LIN {X 0,Y 183.259,Z 699.514,A -85,B 0,C 180,E1 -22058.824,E2 -22058.824} C_VEL
LIN {X 0,Y 184.158,Z 697.784,A -85,B 0,C 180,E1 -22063.237,E2 -22063.237} C_VEL
LIN {X 0,Y 186.021,Z 694.918,A -85,B 0,C 180,E1 -22067.592,E2 -22067.592} C_VEL
LIN {X 0,Y 188.736,Z 690.854,A -85,B 0,C 180,E1 -22071.862,E2 -22071.862} C_VEL
LIN {X 0,Y 192.48,Z 685.477,A -85,B 0,C 180,E1 -22075.986,E2 -22075.986} C_VEL
LIN {X 0,Y 197.248,Z 678.651,A -85,B 0,C 180,E1 -22079.922,E2 -22079.922} C_VEL
LIN {X 0,Y 201.739,Z 671.619,A -85,B 0,C 180,E1 -22083.124,E2 -22083.124} C_VEL
LIN {X 0,Y 207.459,Z 662.596,A -85,B 0,C 180,E1 -22086.359,E2 -22086.359} C_VEL
LIN {X 0,Y 213.578,Z 652.129,A -85,B 0,C 180,E1 -22089.304,E2 -22089.304} C_VEL
LIN {X 0,Y 219.354,Z 641.413,A -85,B 0,C 180,E1 -22091.669,E2 -22091.669} C_VEL
LIN {X 0,Y 225.11,Z 629.438,A -85,B 0,C 180,E1 -22093.775,E2 -22093.775} C_VEL
LIN {X 0,Y 229.636,Z 618.5,A -85,B 0,C 180,E1 -22095.362,E2 -22095.362} C_VEL
LIN {X 0,Y 234.673,Z 604.884,A -85,B 0,C 180,E1 -22096.885,E2 -22096.885} C_VEL
LIN {X 0,Y 238.03,Z 593.851,A -85,B 0,C 180,E1 -22097.888,E2 -22097.888} C_VEL
LIN {X 0,Y 241.922,Z 578.93,A -85,B 0,C 180,E1 -22098.895,E2 -22098.895} C_VEL
LIN {X 0,Y 244.786,Z 564.165,A -85,B 0,C 180,E1 -22099.617,E2 -22099.617} C_VEL
LIN {X 0,Y 246.64,Z 549.204,A -85,B 0,C 180,E1 -22100.137,E2 -22100.137} C_VEL
LIN {X 0,Y 251.554,Z 483.18,A -85,B 0,C 180,E1 -22101.823,E2 -22101.823} C_VEL
LIN {X 0,Y 246.033,Z 470.679,A -85,B 0,C 180,E1 -22104.466,E2 -22104.466} C_VEL
LIN {X 0,Y 241.017,Z 460.608,A -85,B 0,C 180,E1 -22107.097,E2 -22107.097} C_VEL
LIN {X 0,Y 236.074,Z 451.47,A -85,B 0,C 180,E1 -22110.005,E2 -22110.005} C_VEL
LIN {X 0,Y 233.032,Z 446.227,A -85,B 0,C 180,E1 -22112.006,E2 -22112.006} C_VEL
LIN {X 0,Y 229.878,Z 441.234,A -85,B 0,C 180,E1 -22114.295,E2 -22114.295} C_VEL
LIN {X 0,Y 227.435,Z 437.174,A -85,B 0,C 180,E1 -22116.315,E2 -22116.315} C_VEL
LIN {X 0,Y 223.91,Z 432.279,A -85,B 0,C 180,E1 -22119.657,E2 -22119.657} C_VEL
LIN {X 0,Y 221.334,Z 429.386,A -85,B 0,C 180,E1 -22122.645,E2 -22122.645} C_VEL
LIN {X 0,Y 220.368,Z 427.276,A -85,B 0,C 180,E1 -22124.153,E2 -22124.153} C_VEL
LIN {X 0,Y 217.435,Z 424.585,A -85,B 0,C 180,E1 -22130.019,E2 -22130.019} C_VEL
LIN {X 0,Y 216.873,Z 422.233,A -85,B 0,C 180,E1 -22133.722,E2 -22133.722} C_VEL
LIN {X 0,Y 217.021,Z 422.113,A -85,B 0,C 180,E1 -22137.712,E2 -22137.712} C_VEL
LIN {X 0,Y 218.644,Z 426.038,A -85,B 0,C 180,E1 -22143.478,E2 -22143.478} C_VEL
LIN {X 0,Y 220.595,Z 427.431,A -85,B 0,C 180,E1 -22146.633,E2 -22146.633} C_VEL
LIN {X 0,Y 222.451,Z 430.766,A -85,B 0,C 180,E1 -22149.219,E2 -22149.219} C_VEL
LIN {X 0,Y 224.481,Z 432.884,A -85,B 0,C 180,E1 -22151.385,E2 -22151.385} C_VEL
LIN {X 0,Y 227.136,Z 436.564,A -85,B 0,C 180,E1 -22153.876,E2 -22153.876} C_VEL
LIN {X 0,Y 228.488,Z 438.495,A -85,B 0,C 180,E1 -22155.014,E2 -22155.014} C_VEL
LIN {X 0,Y 231.327,Z 442.468,A -85,B 0,C 180,E1 -22157.174,E2 -22157.174} C_VEL
LIN {X 0,Y 234.852,Z 447.543,A -85,B 0,C 180,E1 -22159.553,E2 -22159.553} C_VEL
LIN {X 0,Y 239.256,Z 453.973,A -85,B 0,C 180,E1 -22162.166,E2 -22162.166} C_VEL
LIN {X 0,Y 245.737,Z 464.47,A -85,B 0,C 180,E1 -22165.541,E2 -22165.541} C_VEL
LIN {X 0,Y 250.868,Z 473.742,A -85,B 0,C 180,E1 -22167.93,E2 -22167.93} C_VEL
LIN {X 0,Y 251.979,Z 476.143,A -85,B 0,C 180,E1 -22168.434,E2 -22168.434} C_VEL
LIN {X 0,Y 247.582,Z 533.829,A -85,B 0,C 180,E1 -22169.849,E2 -22169.849} C_VEL
LIN {X 0,Y 246.025,Z 550.183,A -85,B 0,C 180,E1 -22170.374,E2 -22170.374} C_VEL
LIN {X 0,Y 243.766,Z 564.236,A -85,B 0,C 180,E1 -22171.029,E2 -22171.029} C_VEL
LIN {X 0,Y 240.872,Z 577.724,A -85,B 0,C 180,E1 -22171.905,E2 -22171.905} C_VEL
LIN {X 0,Y 236.947,Z 591.791,A -85,B 0,C 180,E1 -22173.079,E2 -22173.079} C_VEL
LIN {X 0,Y 233.016,Z 603.642,A -85,B 0,C 180,E1 -22174.345,E2 -22174.345} C_VEL
LIN {X 0,Y 227.704,Z 617.399,A -85,B 0,C 180,E1 -22176.242,E2 -22176.242} C_VEL
LIN {X 0,Y 221.933,Z 629.908,A -85,B 0,C 180,E1 -22178.394,E2 -22178.394} C_VEL
LIN {X 0,Y 215.979,Z 641.386,A -85,B 0,C 180,E1 -22180.913,E2 -22180.913} C_VEL
LIN {X 0,Y 210.607,Z 650.717,A -85,B 0,C 180,E1 -22183.464,E2 -22183.464} C_VEL
LIN {X 0,Y 204.838,Z 659.969,A -85,B 0,C 180,E1 -22186.67,E2 -22186.67} C_VEL
LIN {X 0,Y 199.72,Z 667.593,A -85,B 0,C 180,E1 -22190.044,E2 -22190.044} C_VEL
LIN {X 0,Y 195.23,Z 673.844,A -85,B 0,C 180,E1 -22193.56,E2 -22193.56} C_VEL
LIN {X 0,Y 190.825,Z 679.701,A -85,B 0,C 180,E1 -22197.898,E2 -22197.898} C_VEL
LIN {X 0,Y 188.424,Z 682.875,A -85,B 0,C 180,E1 -22200.995,E2 -22200.995} C_VEL
LIN {X 0,Y 185.865,Z 686.124,A -85,B 0,C 180,E1 -22205.422,E2 -22205.422} C_VEL
LIN {X 0,Y 184.12,Z 688.111,A -85,B 0,C 180,E1 -22209.908,E2 -22209.908} C_VEL
LIN {X 0,Y 183.277,Z 688.904,A -85,B 0,C 180,E1 -22214.43,E2 -22214.43} C_VEL
LIN {X 0,Y 182.843,Z 688.545,A -85,B 0,C 180,E1 -22218.92,E2 -22218.92} C_VEL
LIN {X 0,Y 183.06,Z 687.039,A -85,B 0,C 180,E1 -22223.386,E2 -22223.386} C_VEL
LIN {X 0,Y 183.36,Z 685.852,A -85,B 0,C 180,E1 -22225.604,E2 -22225.604} C_VEL
LIN {X 0,Y 183.892,Z 682.596,A -85,B 0,C 180,E1 -22230,E2 -22230} C_VEL
LIN {X 0,Y 185.221,Z 678.05,A -85,B 0,C 180,E1 -22234.352,E2 -22234.352} C_VEL
LIN {X 0,Y 187.182,Z 672.165,A -85,B 0,C 180,E1 -22238.638,E2 -22238.638} C_VEL
LIN {X 0,Y 190.032,Z 664.763,A -85,B 0,C 180,E1 -22242.821,E2 -22242.821} C_VEL
LIN {X 0,Y 193.156,Z 656.84,A -85,B 0,C 180,E1 -22246.379,E2 -22246.379} C_VEL
LIN {X 0,Y 196.913,Z 647.341,A -85,B 0,C 180,E1 -22249.82,E2 -22249.82} C_VEL
LIN {X 0,Y 200.691,Z 637.648,A -85,B 0,C 180,E1 -22252.657,E2 -22252.657} C_VEL
LIN {X 0,Y 204.827,Z 626.148,A -85,B 0,C 180,E1 -22255.398,E2 -22255.398} C_VEL
LIN {X 0,Y 208.966,Z 613.481,A -85,B 0,C 180,E1 -22257.817,E2 -22257.817} C_VEL
LIN {X 0,Y 212.598,Z 600.987,A -85,B 0,C 180,E1 -22259.727,E2 -22259.727} C_VEL
LIN {X 0,Y 215.977,Z 587.405,A -85,B 0,C 180,E1 -22261.376,E2 -22261.376} C_VEL
LIN {X 0,Y 218.792,Z 573.543,A -85,B 0,C 180,E1 -22262.687,E2 -22262.687} C_VEL
LIN {X 0,Y 221.131,Z 558.77,A -85,B 0,C 180,E1 -22263.724,E2 -22263.724} C_VEL
LIN {X 0,Y 222.823,Z 543.551,A -85,B 0,C 180,E1 -22264.455,E2 -22264.455} C_VEL
LIN {X 0,Y 228.065,Z 457.657,A -85,B 0,C 180,E1 -22266.934,E2 -22266.934} C_VEL
LIN {X 0,Y 223.194,Z 447.442,A -85,B 0,C 180,E1 -22268.557,E2 -22268.557} C_VEL
LIN {X 0,Y 216.298,Z 434.861,A -85,B 0,C 180,E1 -22270.971,E2 -22270.971} C_VEL
LIN {X 0,Y 209.237,Z 423.431,A -85,B 0,C 180,E1 -22273.66,E2 -22273.66} C_VEL
LIN {X 0,Y 202.644,Z 414.059,A -85,B 0,C 180,E1 -22276.417,E2 -22276.417} C_VEL
LIN {X 0,Y 199.885,Z 410.222,A -85,B 0,C 180,E1 -22277.672,E2 -22277.672} C_VEL
LIN {X 0,Y 196.906,Z 406.254,A -85,B 0,C 180,E1 -22279.099,E2 -22279.099} C_VEL
LIN {X 0,Y 194.318,Z 402.919,A -85,B 0,C 180,E1 -22280.412,E2 -22280.412} C_VEL
LIN {X 0,Y 193.325,Z 401.554,A -85,B 0,C 180,E1 -22280.942,E2 -22280.942} C_VEL
LIN {X 0,Y 190.775,Z 398.797,A -85,B 0,C 180,E1 -22282.315,E2 -22282.315} C_VEL
LIN {X 0,Y 189.719,Z 396.646,A -85,B 0,C 180,E1 -22282.982,E2 -22282.982} C_VEL
LIN {X 0,Y 187.094,Z 394.663,A -85,B 0,C 180,E1 -22284.473,E2 -22284.473} C_VEL
LIN {X 0,Y 185.803,Z 392.386,A -85,B 0,C 180,E1 -22285.349,E2 -22285.349} C_VEL
LIN {X 0,Y 185.5,Z 390.99,A -85,B 0,C 180,E1 -22285.684,E2 -22285.684} C_VEL
LIN {X 0,Y 185.524,Z 390.96,A -85,B 0,C 180,E1 -22290.609,E2 -22290.609} C_VEL
LIN {X 0,Y 185.547,Z 390.93,A -85,B 0,C 180,E1 -22295.376,E2 -22295.376} C_VEL
LIN {X 0,Y 185.636,Z 390.969,A -85,B 0,C 180,E1 -22301.17,E2 -22301.17} C_VEL
LIN {X 0,Y 185.673,Z 390.975,A -85,B 0,C 180,E1 -22304.634,E2 -22304.634} C_VEL
LIN {X 0,Y 185.89,Z 390.93,A -85,B 0,C 180,E1 -22309.418,E2 -22309.418} C_VEL
LIN {X 0,Y 185.934,Z 390.931,A -85,B 0,C 180,E1 -22313.488,E2 -22313.488} C_VEL
LIN {X 0,Y 186.179,Z 390.916,A -85,B 0,C 180,E1 -22317.836,E2 -22317.836} C_VEL
LIN {X 0,Y 186.383,Z 390.877,A -85,B 0,C 180,E1 -22319.999,E2 -22319.999} C_VEL
LIN {X 0,Y 185.896,Z 390.952,A -85,B 0,C 180,E1 -22324.335,E2 -22324.335} C_VEL
LIN {X 0,Y 185.975,Z 390.929,A -85,B 0,C 180,E1 -22328.693,E2 -22328.693} C_VEL
LIN {X 0,Y 185.711,Z 390.958,A -85,B 0,C 180,E1 -22333.123,E2 -22333.123} C_VEL
LIN {X 0,Y 185.635,Z 390.971,A -85,B 0,C 180,E1 -22338.829,E2 -22338.829} C_VEL
LIN {X 0,Y 185.609,Z 390.984,A -85,B 0,C 180,E1 -22344.018,E2 -22344.018} C_VEL
LIN {X 0,Y 186.38,Z 393.478,A -85,B 0,C 180,E1 -22344.647,E2 -22344.647} C_VEL
LIN {X 0,Y 188.13,Z 395.653,A -85,B 0,C 180,E1 -22345.738,E2 -22345.738} C_VEL
LIN {X 0,Y 189.916,Z 396.943,A -85,B 0,C 180,E1 -22346.733,E2 -22346.733} C_VEL
LIN {X 0,Y 192.005,Z 400.303,A -85,B 0,C 180,E1 -22347.967,E2 -22347.967} C_VEL
LIN {X 0,Y 193.974,Z 402.192,A -85,B 0,C 180,E1 -22348.985,E2 -22348.985} C_VEL
LIN {X 0,Y 196.455,Z 405.732,A -85,B 0,C 180,E1 -22350.277,E2 -22350.277} C_VEL
LIN {X 0,Y 197.925,Z 407.506,A -85,B 0,C 180,E1 -22350.988,E2 -22350.988} C_VEL
LIN {X 0,Y 201.75,Z 412.692,A -85,B 0,C 180,E1 -22352.771,E2 -22352.771} C_VEL
LIN {X 0,Y 206.077,Z 418.936,A -85,B 0,C 180,E1 -22354.653,E2 -22354.653} C_VEL
LIN {X 0,Y 212.934,Z 431.449,A -85,B 0,C 180,E1 -22357.483,E2 -22357.483} C_VEL
LIN {X 0,Y 219.603,Z 445.413,A -85,B 0,C 180,E1 -22360.02,E2 -22360.02} C_VEL
LIN {X 0,Y 224.756,Z 457.578,A -85,B 0,C 180,E1 -22361.869,E2 -22361.869} C_VEL
LIN {X 0,Y 225.403,Z 459.29,A -85,B 0,C 180,E1 -22362.099,E2 -22362.099} C_VEL
LIN {X 0,Y 225.844,Z 462.305,A -85,B 0,C 180,E1 -22362.335,E2 -22362.335} C_VEL
LIN {X 0,Y 225.217,Z 466.845,A -85,B 0,C 180,E1 -22362.381,E2 -22362.381} C_VEL
LIN {X 0,Y 222.038,Z 477.484,A -85,B 0,C 180,E1 -22362.076,E2 -22362.076} C_VEL
LIN {X 0,Y 221.658,Z 480.258,A -85,B 0,C 180,E1 -22362.105,E2 -22362.105} C_VEL
LIN {X 0,Y 217.032,Z 553.649,A -85,B 0,C 180,E1 -22364.264,E2 -22364.264} C_VEL
LIN {X 0,Y 215.049,Z 569.791,A -85,B 0,C 180,E1 -22365.031,E2 -22365.031} C_VEL
LIN {X 0,Y 212.237,Z 585.232,A -85,B 0,C 180,E1 -22366.106,E2 -22366.106} C_VEL
LIN {X 0,Y 209.045,Z 599.111,A -85,B 0,C 180,E1 -22367.422,E2 -22367.422} C_VEL
LIN {X 0,Y 205.475,Z 612.527,A -85,B 0,C 180,E1 -22369.105,E2 -22369.105} C_VEL
LIN {X 0,Y 201.856,Z 623.921,A -85,B 0,C 180,E1 -22370.872,E2 -22370.872} C_VEL
LIN {X 0,Y 197.797,Z 635.793,A -85,B 0,C 180,E1 -22373.159,E2 -22373.159} C_VEL
LIN {X 0,Y 193.573,Z 646.785,A -85,B 0,C 180,E1 -22375.753,E2 -22375.753} C_VEL
LIN {X 0,Y 189.625,Z 656.949,A -85,B 0,C 180,E1 -22378.743,E2 -22378.743} C_VEL
LIN {X 0,Y 185.641,Z 666.861,A -85,B 0,C 180,E1 -22382.37,E2 -22382.37} C_VEL
LIN {X 0,Y 182.276,Z 675.104,A -85,B 0,C 180,E1 -22386.118,E2 -22386.118} C_VEL
LIN {X 0,Y 179.877,Z 681.389,A -85,B 0,C 180,E1 -22389.668,E2 -22389.668} C_VEL
LIN {X 0,Y 177.864,Z 687.458,A -85,B 0,C 180,E1 -22393.943,E2 -22393.943} C_VEL
LIN {X 0,Y 176.556,Z 692.457,A -85,B 0,C 180,E1 -22398.52,E2 -22398.52} C_VEL
LIN {X 0,Y 176.035,Z 696.126,A -85,B 0,C 180,E1 -22403.121,E2 -22403.121} C_VEL
LIN {X 0,Y 176.019,Z 698.545,A -85,B 0,C 180,E1 -22407.712,E2 -22407.712} C_VEL
LIN {X 0,Y 176.131,Z 699.306,A -85,B 0,C 180,E1 -22410,E2 -22410} C_VEL
LIN {X 0,Y 175.936,Z 699.898,A -85,B 0,C 180,E1 -22414.582,E2 -22414.582} C_VEL
LIN {X 0,Y 176.214,Z 699.33,A -85,B 0,C 180,E1 -22419.18,E2 -22419.18} C_VEL
LIN {X 0,Y 177.194,Z 697.647,A -85,B 0,C 180,E1 -22423.767,E2 -22423.767} C_VEL
LIN {X 0,Y 179.196,Z 694.83,A -85,B 0,C 180,E1 -22428.286,E2 -22428.286} C_VEL
LIN {X 0,Y 182.121,Z 690.816,A -85,B 0,C 180,E1 -22432.699,E2 -22432.699} C_VEL
LIN {X 0,Y 186.067,Z 685.473,A -85,B 0,C 180,E1 -22436.953,E2 -22436.953} C_VEL
LIN {X 0,Y 191.084,Z 678.704,A -85,B 0,C 180,E1 -22440.992,E2 -22440.992} C_VEL
LIN {X 0,Y 196.799,Z 670.339,A -85,B 0,C 180,E1 -22444.847,E2 -22444.847} C_VEL
LIN {X 0,Y 202.654,Z 661.439,A -85,B 0,C 180,E1 -22447.993,E2 -22447.993} C_VEL
LIN {X 0,Y 208.138,Z 652.404,A -85,B 0,C 180,E1 -22450.541,E2 -22450.541} C_VEL
LIN {X 0,Y 214.113,Z 641.786,A -85,B 0,C 180,E1 -22452.929,E2 -22452.929} C_VEL
LIN {X 0,Y 220.036,Z 629.994,A -85,B 0,C 180,E1 -22455.036,E2 -22455.036} C_VEL
LIN {X 0,Y 224.731,Z 619.14,A -85,B 0,C 180,E1 -22456.644,E2 -22456.644} C_VEL
LIN {X 0,Y 229.904,Z 605.716,A -85,B 0,C 180,E1 -22458.17,E2 -22458.17} C_VEL
LIN {X 0,Y 233.366,Z 594.831,A -85,B 0,C 180,E1 -22459.171,E2 -22459.171} C_VEL
LIN {X 0,Y 237.343,Z 580.285,A -85,B 0,C 180,E1 -22460.178,E2 -22460.178} C_VEL
LIN {X 0,Y 240.466,Z 565.248,A -85,B 0,C 180,E1 -22460.926,E2 -22460.926} C_VEL
LIN {X 0,Y 242.522,Z 549.652,A -85,B 0,C 180,E1 -22461.484,E2 -22461.484} C_VEL
LIN {X 0,Y 247.411,Z 486.673,A -85,B 0,C 180,E1 -22463.089,E2 -22463.089} C_VEL
LIN {X 0,Y 247.105,Z 485.359,A -85,B 0,C 180,E1 -22463.269,E2 -22463.269} C_VEL
LIN {X 0,Y 242.127,Z 473.926,A -85,B 0,C 180,E1 -22465.83,E2 -22465.83} C_VEL
LIN {X 0,Y 237.321,Z 464.186,A -85,B 0,C 180,E1 -22468.542,E2 -22468.542} C_VEL
LIN {X 0,Y 233.344,Z 456.624,A -85,B 0,C 180,E1 -22471.06,E2 -22471.06} C_VEL
LIN {X 0,Y 230.817,Z 452.144,A -85,B 0,C 180,E1 -22472.825,E2 -22472.825} C_VEL
LIN {X 0,Y 227.468,Z 446.57,A -85,B 0,C 180,E1 -22475.425,E2 -22475.425} C_VEL
LIN {X 0,Y 225.593,Z 443.377,A -85,B 0,C 180,E1 -22477.082,E2 -22477.082} C_VEL
LIN {X 0,Y 222.514,Z 438.986,A -85,B 0,C 180,E1 -22480.152,E2 -22480.152} C_VEL
LIN {X 0,Y 220.034,Z 436.054,A -85,B 0,C 180,E1 -22483.18,E2 -22483.18} C_VEL
LIN {X 0,Y 219.112,Z 434.167,A -85,B 0,C 180,E1 -22484.674,E2 -22484.674} C_VEL
LIN {X 0,Y 216.43,Z 431.406,A -85,B 0,C 180,E1 -22490.486,E2 -22490.486} C_VEL
LIN {X 0,Y 215.965,Z 429.13,A -85,B 0,C 180,E1 -22494.398,E2 -22494.398} C_VEL
LIN {X 0,Y 216.147,Z 429.172,A -85,B 0,C 180,E1 -22497.703,E2 -22497.703} C_VEL
LIN {X 0,Y 217.54,Z 432.906,A -85,B 0,C 180,E1 -22503.028,E2 -22503.028} C_VEL
LIN {X 0,Y 219.466,Z 434.461,A -85,B 0,C 180,E1 -22506.321,E2 -22506.321} C_VEL
LIN {X 0,Y 221.456,Z 437.897,A -85,B 0,C 180,E1 -22509.131,E2 -22509.131} C_VEL
LIN {X 0,Y 223.066,Z 439.594,A -85,B 0,C 180,E1 -22510.898,E2 -22510.898} C_VEL
LIN {X 0,Y 225.595,Z 443.212,A -85,B 0,C 180,E1 -22513.37,E2 -22513.37} C_VEL
LIN {X 0,Y 229.559,Z 449.003,A -85,B 0,C 180,E1 -22516.623,E2 -22516.623} C_VEL
LIN {X 0,Y 233.234,Z 454.435,A -85,B 0,C 180,E1 -22519.187,E2 -22519.187} C_VEL
LIN {X 0,Y 238.216,Z 462.153,A -85,B 0,C 180,E1 -22522.211,E2 -22522.211} C_VEL
LIN {X 0,Y 243.893,Z 471.728,A -85,B 0,C 180,E1 -22525.225,E2 -22525.225} C_VEL
LIN {X 0,Y 247.906,Z 479.45,A -85,B 0,C 180,E1 -22527.175,E2 -22527.175} C_VEL
LIN {X 0,Y 242.697,Z 544.089,A -85,B 0,C 180,E1 -22528.784,E2 -22528.784} C_VEL
LIN {X 0,Y 240.794,Z 558.358,A -85,B 0,C 180,E1 -22529.38,E2 -22529.38} C_VEL
LIN {X 0,Y 238.341,Z 570.495,A -85,B 0,C 180,E1 -22530.021,E2 -22530.021} C_VEL
LIN {X 0,Y 234.86,Z 584.57,A -85,B 0,C 180,E1 -22531.065,E2 -22531.065} C_VEL
LIN {X 0,Y 230.657,Z 597.71,A -85,B 0,C 180,E1 -22532.271,E2 -22532.271} C_VEL
LIN {X 0,Y 226.085,Z 610.289,A -85,B 0,C 180,E1 -22533.813,E2 -22533.813} C_VEL
LIN {X 0,Y 220.689,Z 622.733,A -85,B 0,C 180,E1 -22535.702,E2 -22535.702} C_VEL
LIN {X 0,Y 215.377,Z 633.328,A -85,B 0,C 180,E1 -22537.692,E2 -22537.692} C_VEL
LIN {X 0,Y 209.369,Z 644.094,A -85,B 0,C 180,E1 -22540.212,E2 -22540.212} C_VEL
LIN {X 0,Y 203.799,Z 653.166,A -85,B 0,C 180,E1 -22542.878,E2 -22542.878} C_VEL
LIN {X 0,Y 197.897,Z 662.027,A -85,B 0,C 180,E1 -22546.171,E2 -22546.171} C_VEL
LIN {X 0,Y 192.327,Z 669.787,A -85,B 0,C 180,E1 -22549.889,E2 -22549.889} C_VEL
LIN {X 0,Y 188.113,Z 675.358,A -85,B 0,C 180,E1 -22553.29,E2 -22553.29} C_VEL
LIN {X 0,Y 183.754,Z 680.742,A -85,B 0,C 180,E1 -22557.625,E2 -22557.625} C_VEL
LIN {X 0,Y 180.46,Z 684.708,A -85,B 0,C 180,E1 -22562.138,E2 -22562.138} C_VEL
LIN {X 0,Y 178.096,Z 687.378,A -85,B 0,C 180,E1 -22566.758,E2 -22566.758} C_VEL
LIN {X 0,Y 176.668,Z 688.829,A -85,B 0,C 180,E1 -22571.443,E2 -22571.443} C_VEL
LIN {X 0,Y 175.939,Z 689.107,A -85,B 0,C 180,E1 -22576.133,E2 -22576.133} C_VEL
LIN {X 0,Y 175.751,Z 688.24,A -85,B 0,C 180,E1 -22580.796,E2 -22580.796} C_VEL
LIN {X 0,Y 176.265,Z 686.216,A -85,B 0,C 180,E1 -22585.426,E2 -22585.426} C_VEL
LIN {X 0,Y 176.801,Z 682.995,A -85,B 0,C 180,E1 -22590,E2 -22590} C_VEL
LIN {X 0,Y 178.145,Z 678.518,A -85,B 0,C 180,E1 -22594.526,E2 -22594.526} C_VEL
LIN {X 0,Y 180.187,Z 672.707,A -85,B 0,C 180,E1 -22598.976,E2 -22598.976} C_VEL
LIN {X 0,Y 183.156,Z 665.384,A -85,B 0,C 180,E1 -22603.311,E2 -22603.311} C_VEL
LIN {X 0,Y 186.386,Z 657.551,A -85,B 0,C 180,E1 -22606.991,E2 -22606.991} C_VEL
LIN {X 0,Y 190.283,Z 648.154,A -85,B 0,C 180,E1 -22610.541,E2 -22610.541} C_VEL
LIN {X 0,Y 194.201,Z 638.579,A -85,B 0,C 180,E1 -22613.459,E2 -22613.459} C_VEL
LIN {X 0,Y 198.514,Z 627.216,A -85,B 0,C 180,E1 -22616.266,E2 -22616.266} C_VEL
LIN {X 0,Y 202.767,Z 614.73,A -85,B 0,C 180,E1 -22618.745,E2 -22618.745} C_VEL
LIN {X 0,Y 206.528,Z 602.463,A -85,B 0,C 180,E1 -22620.693,E2 -22620.693} C_VEL
LIN {X 0,Y 210.015,Z 589.184,A -85,B 0,C 180,E1 -22622.373,E2 -22622.373} C_VEL
LIN {X 0,Y 213.143,Z 574.522,A -85,B 0,C 180,E1 -22623.809,E2 -22623.809} C_VEL
LIN {X 0,Y 215.691,Z 559.161,A -85,B 0,C 180,E1 -22624.908,E2 -22624.908} C_VEL
LIN {X 0,Y 217.464,Z 543.716,A -85,B 0,C 180,E1 -22625.66,E2 -22625.66} C_VEL
LIN {X 0,Y 222.747,Z 459.889,A -85,B 0,C 180,E1 -22628.117,E2 -22628.117} C_VEL
LIN {X 0,Y 216.264,Z 446.755,A -85,B 0,C 180,E1 -22630.416,E2 -22630.416} C_VEL
LIN {X 0,Y 209.578,Z 434.978,A -85,B 0,C 180,E1 -22632.957,E2 -22632.957} C_VEL
LIN {X 0,Y 203.041,Z 424.771,A -85,B 0,C 180,E1 -22635.672,E2 -22635.672} C_VEL
LIN {X 0,Y 196.873,Z 415.972,A -85,B 0,C 180,E1 -22638.512,E2 -22638.512} C_VEL
LIN {X 0,Y 194.039,Z 412.137,A -85,B 0,C 180,E1 -22639.935,E2 -22639.935} C_VEL
LIN {X 0,Y 191.292,Z 408.382,A -85,B 0,C 180,E1 -22641.411,E2 -22641.411} C_VEL
LIN {X 0,Y 187.894,Z 404.332,A -85,B 0,C 180,E1 -22643.339,E2 -22643.339} C_VEL
LIN {X 0,Y 186.966,Z 402.83,A -85,B 0,C 180,E1 -22643.926,E2 -22643.926} C_VEL
LIN {X 0,Y 184.359,Z 400.333,A -85,B 0,C 180,E1 -22645.529,E2 -22645.529} C_VEL
LIN {X 0,Y 182.819,Z 397.553,A -85,B 0,C 180,E1 -22646.646,E2 -22646.646} C_VEL
LIN {X 0,Y 180.24,Z 395.757,A -85,B 0,C 180,E1 -22648.4,E2 -22648.4} C_VEL
LIN {X 0,Y 178.789,Z 393.322,A -85,B 0,C 180,E1 -22649.595,E2 -22649.595} C_VEL
LIN {X 0,Y 178.466,Z 391.85,A -85,B 0,C 180,E1 -22650.039,E2 -22650.039} C_VEL
LIN {X 0,Y 178.466,Z 391.806,A -85,B 0,C 180,E1 -22654.924,E2 -22654.924} C_VEL
LIN {X 0,Y 178.567,Z 391.853,A -85,B 0,C 180,E1 -22660.838,E2 -22660.838} C_VEL
LIN {X 0,Y 178.647,Z 391.848,A -85,B 0,C 180,E1 -22666.346,E2 -22666.346} C_VEL
LIN {X 0,Y 178.908,Z 391.816,A -85,B 0,C 180,E1 -22670.959,E2 -22670.959} C_VEL
LIN {X 0,Y 179.126,Z 391.793,A -85,B 0,C 180,E1 -22677.75,E2 -22677.75} C_VEL
LIN {X 0,Y 179.348,Z 391.752,A -85,B 0,C 180,E1 -22679.999,E2 -22679.999} C_VEL
LIN {X 0,Y 178.845,Z 391.832,A -85,B 0,C 180,E1 -22684.507,E2 -22684.507} C_VEL
LIN {X 0,Y 178.906,Z 391.811,A -85,B 0,C 180,E1 -22689.04,E2 -22689.04} C_VEL
LIN {X 0,Y 178.638,Z 391.839,A -85,B 0,C 180,E1 -22693.653,E2 -22693.653} C_VEL
LIN {X 0,Y 178.592,Z 391.85,A -85,B 0,C 180,E1 -22699.185,E2 -22699.185} C_VEL
LIN {X 0,Y 178.574,Z 392.022,A -85,B 0,C 180,E1 -22699.733,E2 -22699.733} C_VEL
LIN {X 0,Y 179.394,Z 394.516,A -85,B 0,C 180,E1 -22700.528,E2 -22700.528} C_VEL
LIN {X 0,Y 181.242,Z 396.619,A -85,B 0,C 180,E1 -22701.914,E2 -22701.914} C_VEL
LIN {X 0,Y 183.149,Z 397.908,A -85,B 0,C 180,E1 -22703.177,E2 -22703.177} C_VEL
LIN {X 0,Y 184.87,Z 400.948,A -85,B 0,C 180,E1 -22704.401,E2 -22704.401} C_VEL
LIN {X 0,Y 187.517,Z 403.423,A -85,B 0,C 180,E1 -22705.997,E2 -22705.997} C_VEL
LIN {X 0,Y 189.975,Z 406.954,A -85,B 0,C 180,E1 -22707.468,E2 -22707.468} C_VEL
LIN {X 0,Y 191.456,Z 408.616,A -85,B 0,C 180,E1 -22708.278,E2 -22708.278} C_VEL
LIN {X 0,Y 194.443,Z 412.472,A -85,B 0,C 180,E1 -22709.856,E2 -22709.856} C_VEL
LIN {X 0,Y 200.985,Z 421.656,A -85,B 0,C 180,E1 -22713.004,E2 -22713.004} C_VEL
LIN {X 0,Y 205.596,Z 429.612,A -85,B 0,C 180,E1 -22715.067,E2 -22715.067} C_VEL
LIN {X 0,Y 212.121,Z 442.64,A -85,B 0,C 180,E1 -22717.796,E2 -22717.796} C_VEL
LIN {X 0,Y 218.362,Z 456.878,A -85,B 0,C 180,E1 -22720.218,E2 -22720.218} C_VEL
LIN {X 0,Y 222.385,Z 467.655,A -85,B 0,C 180,E1 -22721.73,E2 -22721.73} C_VEL
LIN {X 0,Y 221.658,Z 480.258,A -85,B 0,C 180,E1 -22722.105,E2 -22722.105} C_VEL
LIN {X 0,Y 220.81,Z 486.102,A -85,B 0,C 180,E1 -22722.155,E2 -22722.155} C_VEL
LIN {X 0,Y 215.427,Z 505.1,A -85,B 0,C 180,E1 -22721.662,E2 -22721.662} C_VEL
LIN {X 0,Y 214.625,Z 510.94,A -85,B 0,C 180,E1 -22721.723,E2 -22721.723} C_VEL
LIN {X 0,Y 211.701,Z 554.012,A -85,B 0,C 180,E1 -22723.014,E2 -22723.014} C_VEL
LIN {X 0,Y 209.647,Z 570.011,A -85,B 0,C 180,E1 -22723.797,E2 -22723.797} C_VEL
LIN {X 0,Y 206.884,Z 584.764,A -85,B 0,C 180,E1 -22724.835,E2 -22724.835} C_VEL
LIN {X 0,Y 203.323,Z 599.611,A -85,B 0,C 180,E1 -22726.265,E2 -22726.265} C_VEL
LIN {X 0,Y 199.572,Z 613.115,A -85,B 0,C 180,E1 -22728.003,E2 -22728.003} C_VEL
LIN {X 0,Y 195.891,Z 624.218,A -85,B 0,C 180,E1 -22729.775,E2 -22729.775} C_VEL
LIN {X 0,Y 191.68,Z 636.005,A -85,B 0,C 180,E1 -22732.11,E2 -22732.11} C_VEL
LIN {X 0,Y 186.927,Z 647.834,A -85,B 0,C 180,E1 -22735.015,E2 -22735.015} C_VEL
LIN {X 0,Y 182.875,Z 657.791,A -85,B 0,C 180,E1 -22738.101,E2 -22738.101} C_VEL
LIN {X 0,Y 178.723,Z 667.521,A -85,B 0,C 180,E1 -22741.843,E2 -22741.843} C_VEL
LIN {X 0,Y 175.265,Z 675.605,A -85,B 0,C 180,E1 -22745.731,E2 -22745.731} C_VEL
LIN {X 0,Y 172.668,Z 682.141,A -85,B 0,C 180,E1 -22749.632,E2 -22749.632} C_VEL
LIN {X 0,Y 170.54,Z 688.457,A -85,B 0,C 180,E1 -22754.462,E2 -22754.462} C_VEL
LIN {X 0,Y 169.315,Z 693.161,A -85,B 0,C 180,E1 -22759.234,E2 -22759.234} C_VEL
LIN {X 0,Y 168.946,Z 695.797,A -85,B 0,C 180,E1 -22762.831,E2 -22762.831} C_VEL
LIN {X 0,Y 168.944,Z 698.267,A -85,B 0,C 180,E1 -22767.616,E2 -22767.616} C_VEL
LIN {X 0,Y 169.038,Z 699.05,A -85,B 0,C 180,E1 -22770,E2 -22770} C_VEL
LIN {X 0,Y 168.846,Z 699.666,A -85,B 0,C 180,E1 -22774.775,E2 -22774.775} C_VEL
LIN {X 0,Y 169.154,Z 699.144,A -85,B 0,C 180,E1 -22779.566,E2 -22779.566} C_VEL
LIN {X 0,Y 170.247,Z 697.509,A -85,B 0,C 180,E1 -22784.341,E2 -22784.341} C_VEL
LIN {X 0,Y 172.401,Z 694.744,A -85,B 0,C 180,E1 -22789.034,E2 -22789.034} C_VEL
LIN {X 0,Y 175.549,Z 690.769,A -85,B 0,C 180,E1 -22793.6,E2 -22793.6} C_VEL
LIN {X 0,Y 179.718,Z 685.47,A -85,B 0,C 180,E1 -22797.987,E2 -22797.987} C_VEL
LIN {X 0,Y 185.003,Z 678.76,A -85,B 0,C 180,E1 -22802.13,E2 -22802.13} C_VEL
LIN {X 0,Y 190.141,Z 671.585,A -85,B 0,C 180,E1 -22805.595,E2 -22805.595} C_VEL
LIN {X 0,Y 196.181,Z 662.98,A -85,B 0,C 180,E1 -22808.823,E2 -22808.823} C_VEL
LIN {X 0,Y 202.807,Z 652.678,A -85,B 0,C 180,E1 -22811.842,E2 -22811.842} C_VEL
LIN {X 0,Y 208.972,Z 642.159,A -85,B 0,C 180,E1 -22814.255,E2 -22814.255} C_VEL
LIN {X 0,Y 215.057,Z 630.566,A -85,B 0,C 180,E1 -22816.358,E2 -22816.358} C_VEL
LIN {X 0,Y 219.944,Z 619.734,A -85,B 0,C 180,E1 -22817.981,E2 -22817.981} C_VEL
LIN {X 0,Y 225.255,Z 606.483,A -85,B 0,C 180,E1 -22819.509,E2 -22819.509} C_VEL
LIN {X 0,Y 229.463,Z 593.865,A -85,B 0,C 180,E1 -22820.656,E2 -22820.656} C_VEL
LIN {X 0,Y 233.558,Z 579.091,A -85,B 0,C 180,E1 -22821.651,E2 -22821.651} C_VEL
LIN {X 0,Y 236.561,Z 564.583,A -85,B 0,C 180,E1 -22822.366,E2 -22822.366} C_VEL
LIN {X 0,Y 238.684,Z 548.69,A -85,B 0,C 180,E1 -22822.919,E2 -22822.919} C_VEL
LIN {X 0,Y 243.461,Z 489.202,A -85,B 0,C 180,E1 -22824.425,E2 -22824.425} C_VEL
LIN {X 0,Y 239.078,Z 478.862,A -85,B 0,C 180,E1 -22826.822,E2 -22826.822} C_VEL
LIN {X 0,Y 234.322,Z 468.788,A -85,B 0,C 180,E1 -22829.691,E2 -22829.691} C_VEL
LIN {X 0,Y 229.79,Z 459.916,A -85,B 0,C 180,E1 -22832.816,E2 -22832.816} C_VEL
LIN {X 0,Y 226.202,Z 453.861,A -85,B 0,C 180,E1 -22835.639,E2 -22835.639} C_VEL
LIN {X 0,Y 223.903,Z 449.779,A -85,B 0,C 180,E1 -22837.752,E2 -22837.752} C_VEL
LIN {X 0,Y 221.048,Z 445.699,A -85,B 0,C 180,E1 -22840.74,E2 -22840.74} C_VEL
LIN {X 0,Y 218.607,Z 442.445,A -85,B 0,C 180,E1 -22843.954,E2 -22843.954} C_VEL
LIN {X 0,Y 217.974,Z 441.083,A -85,B 0,C 180,E1 -22845.053,E2 -22845.053} C_VEL
LIN {X 0,Y 215.461,Z 438.305,A -85,B 0,C 180,E1 -22850.851,E2 -22850.851} C_VEL
LIN {X 0,Y 215.097,Z 436.169,A -85,B 0,C 180,E1 -22854.376,E2 -22854.376} C_VEL
LIN {X 0,Y 215.216,Z 436.145,A -85,B 0,C 180,E1 -22857.256,E2 -22857.256} C_VEL
LIN {X 0,Y 216.652,Z 439.99,A -85,B 0,C 180,E1 -22863.022,E2 -22863.022} C_VEL
LIN {X 0,Y 218.283,Z 441.315,A -85,B 0,C 180,E1 -22865.891,E2 -22865.891} C_VEL
LIN {X 0,Y 220.29,Z 444.813,A -85,B 0,C 180,E1 -22868.833,E2 -22868.833} C_VEL
LIN {X 0,Y 221.644,Z 446.243,A -85,B 0,C 180,E1 -22870.372,E2 -22870.372} C_VEL
LIN {X 0,Y 224.253,Z 450.046,A -85,B 0,C 180,E1 -22873.019,E2 -22873.019} C_VEL
LIN {X 0,Y 227.981,Z 455.804,A -85,B 0,C 180,E1 -22876.195,E2 -22876.195} C_VEL
LIN {X 0,Y 231.312,Z 460.866,A -85,B 0,C 180,E1 -22878.605,E2 -22878.605} C_VEL
LIN {X 0,Y 235.995,Z 468.361,A -85,B 0,C 180,E1 -22881.569,E2 -22881.569} C_VEL
LIN {X 0,Y 241.794,Z 478.53,A -85,B 0,C 180,E1 -22884.77,E2 -22884.77} C_VEL
LIN {X 0,Y 243.885,Z 482.614,A -85,B 0,C 180,E1 -22885.838,E2 -22885.838} C_VEL
LIN {X 0,Y 238.72,Z 544.851,A -85,B 0,C 180,E1 -22887.396,E2 -22887.396} C_VEL
LIN {X 0,Y 236.434,Z 560.647,A -85,B 0,C 180,E1 -22888.06,E2 -22888.06} C_VEL
LIN {X 0,Y 233.695,Z 573.206,A -85,B 0,C 180,E1 -22888.763,E2 -22888.763} C_VEL
LIN {X 0,Y 229.954,Z 587.28,A -85,B 0,C 180,E1 -22889.863,E2 -22889.863} C_VEL
LIN {X 0,Y 225.661,Z 599.916,A -85,B 0,C 180,E1 -22891.078,E2 -22891.078} C_VEL
LIN {X 0,Y 220.802,Z 612.481,A -85,B 0,C 180,E1 -22892.674,E2 -22892.674} C_VEL
LIN {X 0,Y 215.367,Z 624.321,A -85,B 0,C 180,E1 -22894.515,E2 -22894.515} C_VEL
LIN {X 0,Y 209.894,Z 634.75,A -85,B 0,C 180,E1 -22896.524,E2 -22896.524} C_VEL
LIN {X 0,Y 203.686,Z 645.315,A -85,B 0,C 180,E1 -22899.073,E2 -22899.073} C_VEL
LIN {X 0,Y 197.938,Z 654.218,A -85,B 0,C 180,E1 -22901.787,E2 -22901.787} C_VEL
LIN {X 0,Y 191.809,Z 662.932,A -85,B 0,C 180,E1 -22905.144,E2 -22905.144} C_VEL
LIN {X 0,Y 186.511,Z 669.931,A -85,B 0,C 180,E1 -22908.594,E2 -22908.594} C_VEL
LIN {X 0,Y 180.986,Z 676.737,A -85,B 0,C 180,E1 -22912.994,E2 -22912.994} C_VEL
LIN {X 0,Y 176.567,Z 681.831,A -85,B 0,C 180,E1 -22917.497,E2 -22917.497} C_VEL
LIN {X 0,Y 173.958,Z 684.751,A -85,B 0,C 180,E1 -22921,E2 -22921} C_VEL
LIN {X 0,Y 171.368,Z 687.487,A -85,B 0,C 180,E1 -22925.788,E2 -22925.788} C_VEL
LIN {X 0,Y 169.746,Z 689.004,A -85,B 0,C 180,E1 -22930.657,E2 -22930.657} C_VEL
LIN {X 0,Y 168.908,Z 689.346,A -85,B 0,C 180,E1 -22935.543,E2 -22935.543} C_VEL
LIN {X 0,Y 168.655,Z 688.542,A -85,B 0,C 180,E1 -22940.405,E2 -22940.405} C_VEL
LIN {X 0,Y 169.193,Z 686.408,A -85,B 0,C 180,E1 -22945.521,E2 -22945.521} C_VEL
LIN {X 0,Y 169.713,Z 683.393,A -85,B 0,C 180,E1 -22950,E2 -22950} C_VEL
LIN {X 0,Y 171.069,Z 678.987,A -85,B 0,C 180,E1 -22954.713,E2 -22954.713} C_VEL
LIN {X 0,Y 173.201,Z 673.248,A -85,B 0,C 180,E1 -22959.341,E2 -22959.341} C_VEL
LIN {X 0,Y 176.295,Z 666.005,A -85,B 0,C 180,E1 -22963.839,E2 -22963.839} C_VEL
LIN {X 0,Y 179.642,Z 658.261,A -85,B 0,C 180,E1 -22967.65,E2 -22967.65} C_VEL
LIN {X 0,Y 183.688,Z 648.962,A -85,B 0,C 180,E1 -22971.314,E2 -22971.314} C_VEL
LIN {X 0,Y 187.752,Z 639.503,A -85,B 0,C 180,E1 -22974.315,E2 -22974.315} C_VEL
LIN {X 0,Y 192.206,Z 628.279,A -85,B 0,C 180,E1 -22977.198,E2 -22977.198} C_VEL
LIN {X 0,Y 196.624,Z 615.961,A -85,B 0,C 180,E1 -22979.732,E2 -22979.732} C_VEL
LIN {X 0,Y 200.937,Z 602.358,A -85,B 0,C 180,E1 -22981.939,E2 -22981.939} C_VEL
LIN {X 0,Y 204.564,Z 589.009,A -85,B 0,C 180,E1 -22983.641,E2 -22983.641} C_VEL
LIN {X 0,Y 207.805,Z 574.222,A -85,B 0,C 180,E1 -22985.096,E2 -22985.096} C_VEL
LIN {X 0,Y 210.453,Z 558.629,A -85,B 0,C 180,E1 -22986.205,E2 -22986.205} C_VEL
LIN {X 0,Y 212.221,Z 543.464,A -85,B 0,C 180,E1 -22986.941,E2 -22986.941} C_VEL
LIN {X 0,Y 217.573,Z 462.42,A -85,B 0,C 180,E1 -22989.33,E2 -22989.33} C_VEL
LIN {X 0,Y 211.574,Z 450.286,A -85,B 0,C 180,E1 -22991.583,E2 -22991.583} C_VEL
LIN {X 0,Y 205.412,Z 439.302,A -85,B 0,C 180,E1 -22994.068,E2 -22994.068} C_VEL
LIN {X 0,Y 199.651,Z 430.132,A -85,B 0,C 180,E1 -22996.594,E2 -22996.594} C_VEL
LIN {X 0,Y 193.674,Z 421.449,A -85,B 0,C 180,E1 -22999.493,E2 -22999.493} C_VEL
LIN {X 0,Y 190.874,Z 417.615,A -85,B 0,C 180,E1 -23000.977,E2 -23000.977} C_VEL
LIN {X 0,Y 187.82,Z 413.491,A -85,B 0,C 180,E1 -23002.714,E2 -23002.714} C_VEL
LIN {X 0,Y 184.976,Z 409.688,A -85,B 0,C 180,E1 -23004.46,E2 -23004.46} C_VEL
LIN {X 0,Y 181.591,Z 405.801,A -85,B 0,C 180,E1 -23006.691,E2 -23006.691} C_VEL
LIN {X 0,Y 180.552,Z 404.041,A -85,B 0,C 180,E1 -23007.475,E2 -23007.475} C_VEL
LIN {X 0,Y 177.825,Z 401.641,A -85,B 0,C 180,E1 -23009.479,E2 -23009.479} C_VEL
LIN {X 0,Y 176.127,Z 398.552,A -85,B 0,C 180,E1 -23010.999,E2 -23010.999} C_VEL
LIN {X 0,Y 173.253,Z 396.692,A -85,B 0,C 180,E1 -23013.498,E2 -23013.498} C_VEL
LIN {X 0,Y 171.804,Z 394.276,A -85,B 0,C 180,E1 -23015.084,E2 -23015.084} C_VEL
LIN {X 0,Y 171.411,Z 392.691,A -85,B 0,C 180,E1 -23015.723,E2 -23015.723} C_VEL
LIN {X 0,Y 171.521,Z 392.73,A -85,B 0,C 180,E1 -23020.864,E2 -23020.864} C_VEL
LIN {X 0,Y 171.562,Z 392.737,A -85,B 0,C 180,E1 -23025.77,E2 -23025.77} C_VEL
LIN {X 0,Y 171.846,Z 392.689,A -85,B 0,C 180,E1 -23030.584,E2 -23030.584} C_VEL
LIN {X 0,Y 171.786,Z 392.684,A -85,B 0,C 180,E1 -23035.306,E2 -23035.306} C_VEL
LIN {X 0,Y 172.313,Z 392.628,A -85,B 0,C 180,E1 -23039.999,E2 -23039.999} C_VEL
LIN {X 0,Y 171.795,Z 392.711,A -85,B 0,C 180,E1 -23044.692,E2 -23044.692} C_VEL
LIN {X 0,Y 171.844,Z 392.694,A -85,B 0,C 180,E1 -23049.414,E2 -23049.414} C_VEL
LIN {X 0,Y 171.606,Z 392.9,A -85,B 0,C 180,E1 -23054.148,E2 -23054.148} C_VEL
LIN {X 0,Y 172.234,Z 395.051,A -85,B 0,C 180,E1 -23055.001,E2 -23055.001} C_VEL
LIN {X 0,Y 174.231,Z 397.447,A -85,B 0,C 180,E1 -23057.003,E2 -23057.003} C_VEL
LIN {X 0,Y 176.427,Z 398.815,A -85,B 0,C 180,E1 -23058.851,E2 -23058.851} C_VEL
LIN {X 0,Y 177.824,Z 401.579,A -85,B 0,C 180,E1 -23060.116,E2 -23060.116} C_VEL
LIN {X 0,Y 180.406,Z 403.894,A -85,B 0,C 180,E1 -23062.021,E2 -23062.021} C_VEL
LIN {X 0,Y 181.023,Z 404.65,A -85,B 0,C 180,E1 -23062.467,E2 -23062.467} C_VEL
LIN {X 0,Y 183.249,Z 407.935,A -85,B 0,C 180,E1 -23064.046,E2 -23064.046} C_VEL
LIN {X 0,Y 185.203,Z 409.888,A -85,B 0,C 180,E1 -23065.271,E2 -23065.271} C_VEL
LIN {X 0,Y 187.961,Z 413.588,A -85,B 0,C 180,E1 -23066.959,E2 -23066.959} C_VEL
LIN {X 0,Y 189.384,Z 415.569,A -85,B 0,C 180,E1 -23067.786,E2 -23067.786} C_VEL
LIN {X 0,Y 192.559,Z 419.842,A -85,B 0,C 180,E1 -23069.519,E2 -23069.519} C_VEL
LIN {X 0,Y 197.462,Z 426.681,A -85,B 0,C 180,E1 -23071.966,E2 -23071.966} C_VEL
LIN {X 0,Y 202.133,Z 435.038,A -85,B 0,C 180,E1 -23074.175,E2 -23074.175} C_VEL
LIN {X 0,Y 207.662,Z 446.275,A -85,B 0,C 180,E1 -23076.618,E2 -23076.618} C_VEL
LIN {X 0,Y 213.91,Z 460.81,A -85,B 0,C 180,E1 -23079.193,E2 -23079.193} C_VEL
LIN {X 0,Y 217.158,Z 469.626,A -85,B 0,C 180,E1 -23080.487,E2 -23080.487} C_VEL
LIN {X 0,Y 214.625,Z 510.94,A -85,B 0,C 180,E1 -23081.723,E2 -23081.723} C_VEL
LIN {X 0,Y 213.812,Z 516.787,A -85,B 0,C 180,E1 -23081.782,E2 -23081.782} C_VEL
LIN {X 0,Y 208.329,Z 535.781,A -85,B 0,C 180,E1 -23081.232,E2 -23081.232} C_VEL
LIN {X 0,Y 207.442,Z 541.633,A -85,B 0,C 180,E1 -23081.272,E2 -23081.272} C_VEL
LIN {X 0,Y 205.984,Z 558.852,A -85,B 0,C 180,E1 -23081.907,E2 -23081.907} C_VEL
LIN {X 0,Y 203.674,Z 574.076,A -85,B 0,C 180,E1 -23082.749,E2 -23082.749} C_VEL
LIN {X 0,Y 200.523,Z 588.853,A -85,B 0,C 180,E1 -23083.889,E2 -23083.889} C_VEL
LIN {X 0,Y 196.991,Z 602.608,A -85,B 0,C 180,E1 -23085.347,E2 -23085.347} C_VEL
LIN {X 0,Y 192.806,Z 616.35,A -85,B 0,C 180,E1 -23087.242,E2 -23087.242} C_VEL
LIN {X 0,Y 188.204,Z 629.42,A -85,B 0,C 180,E1 -23089.547,E2 -23089.547} C_VEL
LIN {X 0,Y 183.516,Z 641.367,A -85,B 0,C 180,E1 -23092.212,E2 -23092.212} C_VEL
LIN {X 0,Y 178.69,Z 652.621,A -85,B 0,C 180,E1 -23095.366,E2 -23095.366} C_VEL
LIN {X 0,Y 174.216,Z 662.932,A -85,B 0,C 180,E1 -23099.046,E2 -23099.046} C_VEL
LIN {X 0,Y 170.19,Z 671.75,A -85,B 0,C 180,E1 -23102.983,E2 -23102.983} C_VEL
LIN {X 0,Y 166.629,Z 680.004,A -85,B 0,C 180,E1 -23107.691,E2 -23107.691} C_VEL
LIN {X 0,Y 164.09,Z 686.585,A -85,B 0,C 180,E1 -23112.554,E2 -23112.554} C_VEL
LIN {X 0,Y 162.542,Z 691.696,A -85,B 0,C 180,E1 -23117.514,E2 -23117.514} C_VEL
LIN {X 0,Y 161.881,Z 695.469,A -85,B 0,C 180,E1 -23122.516,E2 -23122.516} C_VEL
LIN {X 0,Y 161.863,Z 697.99,A -85,B 0,C 180,E1 -23127.511,E2 -23127.511} C_VEL
LIN {X 0,Y 161.947,Z 698.782,A -85,B 0,C 180,E1 -23130,E2 -23130} C_VEL
LIN {X 0,Y 161.811,Z 699.276,A -85,B 0,C 180,E1 -23132.622,E2 -23132.622} C_VEL
LIN {X 0,Y 161.821,Z 699.336,A -85,B 0,C 180,E1 -23137.486,E2 -23137.486} C_VEL
LIN {X 0,Y 162.613,Z 698.307,A -85,B 0,C 180,E1 -23142.48,E2 -23142.48} C_VEL
LIN {X 0,Y 164.39,Z 696.161,A -85,B 0,C 180,E1 -23147.413,E2 -23147.413} C_VEL
LIN {X 0,Y 167.213,Z 692.726,A -85,B 0,C 180,E1 -23152.385,E2 -23152.385} C_VEL
LIN {X 0,Y 171.09,Z 688.256,A -85,B 0,C 180,E1 -23156.863,E2 -23156.863} C_VEL
LIN {X 0,Y 176.029,Z 682.327,A -85,B 0,C 180,E1 -23161.267,E2 -23161.267} C_VEL
LIN {X 0,Y 181.266,Z 675.916,A -85,B 0,C 180,E1 -23164.882,E2 -23164.882} C_VEL
LIN {X 0,Y 187.018,Z 668.238,A -85,B 0,C 180,E1 -23168.32,E2 -23168.32} C_VEL
LIN {X 0,Y 193.606,Z 659.042,A -85,B 0,C 180,E1 -23171.49,E2 -23171.49} C_VEL
LIN {X 0,Y 199.665,Z 649.72,A -85,B 0,C 180,E1 -23174.042,E2 -23174.042} C_VEL
LIN {X 0,Y 206.742,Z 637.674,A -85,B 0,C 180,E1 -23176.604,E2 -23176.604} C_VEL
LIN {X 0,Y 213.122,Z 624.987,A -85,B 0,C 180,E1 -23178.737,E2 -23178.737} C_VEL
LIN {X 0,Y 218.926,Z 611.945,A -85,B 0,C 180,E1 -23180.395,E2 -23180.395} C_VEL
LIN {X 0,Y 223.769,Z 598.742,A -85,B 0,C 180,E1 -23181.738,E2 -23181.738} C_VEL
LIN {X 0,Y 228.283,Z 584.234,A -85,B 0,C 180,E1 -23182.807,E2 -23182.807} C_VEL
LIN {X 0,Y 231.824,Z 569.196,A -85,B 0,C 180,E1 -23183.637,E2 -23183.637} C_VEL
LIN {X 0,Y 234.398,Z 553.545,A -85,B 0,C 180,E1 -23184.228,E2 -23184.228} C_VEL
LIN {X 0,Y 239.586,Z 492.217,A -85,B 0,C 180,E1 -23185.803,E2 -23185.803} C_VEL
LIN {X 0,Y 235.627,Z 482.695,A -85,B 0,C 180,E1 -23188.131,E2 -23188.131} C_VEL
LIN {X 0,Y 231.254,Z 473.213,A -85,B 0,C 180,E1 -23190.972,E2 -23190.972} C_VEL
LIN {X 0,Y 227.166,Z 465.033,A -85,B 0,C 180,E1 -23194.01,E2 -23194.01} C_VEL
LIN {X 0,Y 224.353,Z 460.074,A -85,B 0,C 180,E1 -23196.382,E2 -23196.382} C_VEL
LIN {X 0,Y 222.488,Z 456.55,A -85,B 0,C 180,E1 -23198.189,E2 -23198.189} C_VEL
LIN {X 0,Y 219.755,Z 452.505,A -85,B 0,C 180,E1 -23201.168,E2 -23201.168} C_VEL
LIN {X 0,Y 217.34,Z 449.081,A -85,B 0,C 180,E1 -23204.528,E2 -23204.528} C_VEL
LIN {X 0,Y 216.876,Z 447.995,A -85,B 0,C 180,E1 -23205.391,E2 -23205.391} C_VEL
LIN {X 0,Y 214.535,Z 445.323,A -85,B 0,C 180,E1 -23211.049,E2 -23211.049} C_VEL
LIN {X 0,Y 214.225,Z 443.239,A -85,B 0,C 180,E1 -23214.353,E2 -23214.353} C_VEL
LIN {X 0,Y 214.339,Z 443.23,A -85,B 0,C 180,E1 -23217.245,E2 -23217.245} C_VEL
LIN {X 0,Y 215.666,Z 446.972,A -85,B 0,C 180,E1 -23222.803,E2 -23222.803} C_VEL
LIN {X 0,Y 217.176,Z 448.298,A -85,B 0,C 180,E1 -23225.572,E2 -23225.572} C_VEL
LIN {X 0,Y 219.131,Z 451.724,A -85,B 0,C 180,E1 -23228.531,E2 -23228.531} C_VEL
LIN {X 0,Y 220.363,Z 453.201,A -85,B 0,C 180,E1 -23229.997,E2 -23229.997} C_VEL
LIN {X 0,Y 223.402,Z 457.809,A -85,B 0,C 180,E1 -23233.141,E2 -23233.141} C_VEL
LIN {X 0,Y 226.471,Z 462.714,A -85,B 0,C 180,E1 -23235.805,E2 -23235.805} C_VEL
LIN {X 0,Y 230.284,Z 468.6,A -85,B 0,C 180,E1 -23238.613,E2 -23238.613} C_VEL
LIN {X 0,Y 234.922,Z 476.591,A -85,B 0,C 180,E1 -23241.6,E2 -23241.6} C_VEL
LIN {X 0,Y 239.5,Z 485.023,A -85,B 0,C 180,E1 -23244.2,E2 -23244.2} C_VEL
LIN {X 0,Y 239.987,Z 485.998,A -85,B 0,C 180,E1 -23244.463,E2 -23244.463} C_VEL
LIN {X 0,Y 234.971,Z 544.803,A -85,B 0,C 180,E1 -23245.937,E2 -23245.937} C_VEL
LIN {X 0,Y 232.607,Z 560.776,A -85,B 0,C 180,E1 -23246.602,E2 -23246.602} C_VEL
LIN {X 0,Y 229.692,Z 573.749,A -85,B 0,C 180,E1 -23247.321,E2 -23247.321} C_VEL
LIN {X 0,Y 225.722,Z 588.113,A -85,B 0,C 180,E1 -23248.446,E2 -23248.446} C_VEL
LIN {X 0,Y 221.36,Z 600.495,A -85,B 0,C 180,E1 -23249.642,E2 -23249.642} C_VEL
LIN {X 0,Y 216.476,Z 612.668,A -85,B 0,C 180,E1 -23251.184,E2 -23251.184} C_VEL
LIN {X 0,Y 210.729,Z 624.782,A -85,B 0,C 180,E1 -23253.076,E2 -23253.076} C_VEL
LIN {X 0,Y 204.53,Z 636.087,A -85,B 0,C 180,E1 -23255.283,E2 -23255.283} C_VEL
LIN {X 0,Y 198.1,Z 646.534,A -85,B 0,C 180,E1 -23257.874,E2 -23257.874} C_VEL
LIN {X 0,Y 192.059,Z 655.412,A -85,B 0,C 180,E1 -23260.678,E2 -23260.678} C_VEL
LIN {X 0,Y 185.769,Z 663.836,A -85,B 0,C 180,E1 -23264.044,E2 -23264.044} C_VEL
LIN {X 0,Y 179.604,Z 671.487,A -85,B 0,C 180,E1 -23268.031,E2 -23268.031} C_VEL
LIN {X 0,Y 175.114,Z 676.67,A -85,B 0,C 180,E1 -23271.532,E2 -23271.532} C_VEL
LIN {X 0,Y 170.303,Z 681.911,A -85,B 0,C 180,E1 -23276.24,E2 -23276.24} C_VEL
LIN {X 0,Y 167.525,Z 684.794,A -85,B 0,C 180,E1 -23279.773,E2 -23279.773} C_VEL
LIN {X 0,Y 164.68,Z 687.598,A -85,B 0,C 180,E1 -23284.738,E2 -23284.738} C_VEL
LIN {X 0,Y 162.838,Z 689.18,A -85,B 0,C 180,E1 -23289.801,E2 -23289.801} C_VEL
LIN {X 0,Y 161.873,Z 689.586,A -85,B 0,C 180,E1 -23294.9,E2 -23294.9} C_VEL
LIN {X 0,Y 161.538,Z 688.843,A -85,B 0,C 180,E1 -23299.978,E2 -23299.978} C_VEL
LIN {X 0,Y 161.966,Z 686.899,A -85,B 0,C 180,E1 -23305.022,E2 -23305.022} C_VEL
LIN {X 0,Y 162.624,Z 683.789,A -85,B 0,C 180,E1 -23310,E2 -23310} C_VEL
LIN {X 0,Y 163.994,Z 679.452,A -85,B 0,C 180,E1 -23314.917,E2 -23314.917} C_VEL
LIN {X 0,Y 166.224,Z 673.784,A -85,B 0,C 180,E1 -23319.737,E2 -23319.737} C_VEL
LIN {X 0,Y 169.422,Z 666.62,A -85,B 0,C 180,E1 -23324.412,E2 -23324.412} C_VEL
LIN {X 0,Y 172.924,Z 658.962,A -85,B 0,C 180,E1 -23328.36,E2 -23328.36} C_VEL
LIN {X 0,Y 177.13,Z 649.764,A -85,B 0,C 180,E1 -23332.144,E2 -23332.144} C_VEL
LIN {X 0,Y 181.349,Z 640.417,A -85,B 0,C 180,E1 -23335.233,E2 -23335.233} C_VEL
LIN {X 0,Y 185.963,Z 629.316,A -85,B 0,C 180,E1 -23338.191,E2 -23338.191} C_VEL
LIN {X 0,Y 190.544,Z 617.152,A -85,B 0,C 180,E1 -23340.782,E2 -23340.782} C_VEL
LIN {X 0,Y 195.013,Z 603.783,A -85,B 0,C 180,E1 -23343.031,E2 -23343.031} C_VEL
LIN {X 0,Y 198.758,Z 590.651,A -85,B 0,C 180,E1 -23344.762,E2 -23344.762} C_VEL
LIN {X 0,Y 202.126,Z 576.279,A -85,B 0,C 180,E1 -23346.235,E2 -23346.235} C_VEL
LIN {X 0,Y 204.846,Z 561.418,A -85,B 0,C 180,E1 -23347.361,E2 -23347.361} C_VEL
LIN {X 0,Y 206.806,Z 546.182,A -85,B 0,C 180,E1 -23348.165,E2 -23348.165} C_VEL
LIN {X 0,Y 209.034,Z 515.569,A -85,B 0,C 180,E1 -23349.133,E2 -23349.133} C_VEL
LIN {X 0,Y 212.426,Z 464.89,A -85,B 0,C 180,E1 -23350.624,E2 -23350.624} C_VEL
LIN {X 0,Y 206.47,Z 452.802,A -85,B 0,C 180,E1 -23353.015,E2 -23353.015} C_VEL
LIN {X 0,Y 200.148,Z 441.588,A -85,B 0,C 180,E1 -23355.757,E2 -23355.757} C_VEL
LIN {X 0,Y 193.615,Z 431.376,A -85,B 0,C 180,E1 -23358.888,E2 -23358.888} C_VEL
LIN {X 0,Y 188.802,Z 424.288,A -85,B 0,C 180,E1 -23361.48,E2 -23361.48} C_VEL
LIN {X 0,Y 185.062,Z 419.318,A -85,B 0,C 180,E1 -23363.686,E2 -23363.686} C_VEL
LIN {X 0,Y 181.882,Z 415.088,A -85,B 0,C 180,E1 -23365.756,E2 -23365.756} C_VEL
LIN {X 0,Y 179.152,Z 411.682,A -85,B 0,C 180,E1 -23367.689,E2 -23367.689} C_VEL
LIN {X 0,Y 178.394,Z 410.474,A -85,B 0,C 180,E1 -23368.284,E2 -23368.284} C_VEL
LIN {X 0,Y 175.73,Z 407.859,A -85,B 0,C 180,E1 -23370.364,E2 -23370.364} C_VEL
LIN {X 0,Y 174.251,Z 405.201,A -85,B 0,C 180,E1 -23371.751,E2 -23371.751} C_VEL
LIN {X 0,Y 171.529,Z 403.202,A -85,B 0,C 180,E1 -23374.258,E2 -23374.258} C_VEL
LIN {X 0,Y 169.876,Z 400.232,A -85,B 0,C 180,E1 -23376.21,E2 -23376.21} C_VEL
LIN {X 0,Y 169.671,Z 399.608,A -85,B 0,C 180,E1 -23376.503,E2 -23376.503} C_VEL
LIN {X 0,Y 166.779,Z 398.072,A -85,B 0,C 180,E1 -23380.106,E2 -23380.106} C_VEL
LIN {X 0,Y 164.986,Z 395.495,A -85,B 0,C 180,E1 -23383.288,E2 -23383.288} C_VEL
LIN {X 0,Y 164.476,Z 393.615,A -85,B 0,C 180,E1 -23384.827,E2 -23384.827} C_VEL
LIN {X 0,Y 164.767,Z 393.566,A -85,B 0,C 180,E1 -23390.175,E2 -23390.175} C_VEL
LIN {X 0,Y 164.823,Z 393.568,A -85,B 0,C 180,E1 -23392.65,E2 -23392.65} C_VEL
LIN {X 0,Y 165.277,Z 393.503,A -85,B 0,C 180,E1 -23399.999,E2 -23399.999} C_VEL
LIN {X 0,Y 164.769,Z 393.63,A -85,B 0,C 180,E1 -23405.506,E2 -23405.506} C_VEL
LIN {X 0,Y 165.317,Z 395.449,A -85,B 0,C 180,E1 -23406.866,E2 -23406.866} C_VEL
LIN {X 0,Y 167.072,Z 397.988,A -85,B 0,C 180,E1 -23409.871,E2 -23409.871} C_VEL
LIN {X 0,Y 169.853,Z 399.812,A -85,B 0,C 180,E1 -23413.305,E2 -23413.305} C_VEL
LIN {X 0,Y 171.116,Z 402.506,A -85,B 0,C 180,E1 -23414.873,E2 -23414.873} C_VEL
LIN {X 0,Y 173.371,Z 404.704,A -85,B 0,C 180,E1 -23417.09,E2 -23417.09} C_VEL
LIN {X 0,Y 174.465,Z 405.423,A -85,B 0,C 180,E1 -23418.039,E2 -23418.039} C_VEL
LIN {X 0,Y 176.4,Z 408.658,A -85,B 0,C 180,E1 -23419.794,E2 -23419.794} C_VEL
LIN {X 0,Y 178.802,Z 410.94,A -85,B 0,C 180,E1 -23421.622,E2 -23421.622} C_VEL
LIN {X 0,Y 181.336,Z 414.544,A -85,B 0,C 180,E1 -23423.481,E2 -23423.481} C_VEL
LIN {X 0,Y 182.831,Z 416.15,A -85,B 0,C 180,E1 -23424.464,E2 -23424.464} C_VEL
LIN {X 0,Y 186.638,Z 421.372,A -85,B 0,C 180,E1 -23426.863,E2 -23426.863} C_VEL
LIN {X 0,Y 190.674,Z 427.006,A -85,B 0,C 180,E1 -23429.157,E2 -23429.157} C_VEL
LIN {X 0,Y 194.932,Z 433.31,A -85,B 0,C 180,E1 -23431.366,E2 -23431.366} C_VEL
LIN {X 0,Y 200.07,Z 443.061,A -85,B 0,C 180,E1 -23433.893,E2 -23433.893} C_VEL
LIN {X 0,Y 205.609,Z 455.26,A -85,B 0,C 180,E1 -23436.434,E2 -23436.434} C_VEL
LIN {X 0,Y 210.091,Z 466.344,A -85,B 0,C 180,E1 -23438.369,E2 -23438.369} C_VEL
LIN {X 0,Y 212.108,Z 471.806,A -85,B 0,C 180,E1 -23439.215,E2 -23439.215} C_VEL
LIN {X 0,Y 207.442,Z 541.633,A -85,B 0,C 180,E1 -23441.272,E2 -23441.272} C_VEL
LIN {X 0,Y 206.537,Z 547.474,A -85,B 0,C 180,E1 -23441.319,E2 -23441.319} C_VEL
LIN {X 0,Y 203.584,Z 556.924,A -85,B 0,C 180,E1 -23441.119,E2 -23441.119} C_VEL
LIN {X 0,Y 200.294,Z 566.278,A -85,B 0,C 180,E1 -23441.012,E2 -23441.012} C_VEL
LIN {X 0,Y 198.878,Z 571.967,A -85,B 0,C 180,E1 -23441.231,E2 -23441.231} C_VEL
LIN {X 0,Y 195.935,Z 586.11,A -85,B 0,C 180,E1 -23442.285,E2 -23442.285} C_VEL
LIN {X 0,Y 192.659,Z 598.797,A -85,B 0,C 180,E1 -23443.534,E2 -23443.534} C_VEL
LIN {X 0,Y 188.632,Z 612.338,A -85,B 0,C 180,E1 -23445.312,E2 -23445.312} C_VEL
LIN {X 0,Y 184.664,Z 623.49,A -85,B 0,C 180,E1 -23447.133,E2 -23447.133} C_VEL
LIN {X 0,Y 180.049,Z 635.319,A -85,B 0,C 180,E1 -23449.538,E2 -23449.538} C_VEL
LIN {X 0,Y 175.322,Z 646.288,A -85,B 0,C 180,E1 -23452.315,E2 -23452.315} C_VEL
LIN {X 0,Y 170.676,Z 656.595,A -85,B 0,C 180,E1 -23455.596,E2 -23455.596} C_VEL
LIN {X 0,Y 166.208,Z 666.32,A -85,B 0,C 180,E1 -23459.508,E2 -23459.508} C_VEL
LIN {X 0,Y 162.228,Z 674.539,A -85,B 0,C 180,E1 -23463.637,E2 -23463.637} C_VEL
LIN {X 0,Y 159.114,Z 681.487,A -85,B 0,C 180,E1 -23468.056,E2 -23468.056} C_VEL
LIN {X 0,Y 156.739,Z 687.595,A -85,B 0,C 180,E1 -23473.055,E2 -23473.055} C_VEL
LIN {X 0,Y 155.302,Z 692.397,A -85,B 0,C 180,E1 -23478.25,E2 -23478.25} C_VEL
LIN {X 0,Y 154.795,Z 695.137,A -85,B 0,C 180,E1 -23482.171,E2 -23482.171} C_VEL
LIN {X 0,Y 154.773,Z 697.703,A -85,B 0,C 180,E1 -23487.397,E2 -23487.397} C_VEL
LIN {X 0,Y 154.858,Z 698.504,A -85,B 0,C 180,E1 -23490,E2 -23490} C_VEL
LIN {X 0,Y 154.668,Z 699.203,A -85,B 0,C 180,E1 -23495.214,E2 -23495.214} C_VEL
LIN {X 0,Y 155.101,Z 698.777,A -85,B 0,C 180,E1 -23500.442,E2 -23500.442} C_VEL
LIN {X 0,Y 156.421,Z 697.239,A -85,B 0,C 180,E1 -23505.639,E2 -23505.639} C_VEL
LIN {X 0,Y 158.922,Z 694.566,A -85,B 0,C 180,E1 -23510.719,E2 -23510.719} C_VEL
LIN {X 0,Y 162.518,Z 690.653,A -85,B 0,C 180,E1 -23515.623,E2 -23515.623} C_VEL
LIN {X 0,Y 167.222,Z 685.465,A -85,B 0,C 180,E1 -23520.287,E2 -23520.287} C_VEL
LIN {X 0,Y 173.094,Z 678.875,A -85,B 0,C 180,E1 -23524.641,E2 -23524.641} C_VEL
LIN {X 0,Y 178.825,Z 671.739,A -85,B 0,C 180,E1 -23528.295,E2 -23528.295} C_VEL
LIN {X 0,Y 185.304,Z 663.378,A -85,B 0,C 180,E1 -23531.584,E2 -23531.584} C_VEL
LIN {X 0,Y 192.489,Z 653.247,A -85,B 0,C 180,E1 -23534.655,E2 -23534.655} C_VEL
LIN {X 0,Y 199.073,Z 642.933,A -85,B 0,C 180,E1 -23537.101,E2 -23537.101} C_VEL
LIN {X 0,Y 205.991,Z 630.715,A -85,B 0,C 180,E1 -23539.35,E2 -23539.35} C_VEL
LIN {X 0,Y 210.74,Z 620.901,A -85,B 0,C 180,E1 -23540.838,E2 -23540.838} C_VEL
LIN {X 0,Y 216.379,Z 608.004,A -85,B 0,C 180,E1 -23542.345,E2 -23542.345} C_VEL
LIN {X 0,Y 220.804,Z 595.886,A -85,B 0,C 180,E1 -23543.483,E2 -23543.483} C_VEL
LIN {X 0,Y 225.082,Z 581.875,A -85,B 0,C 180,E1 -23544.467,E2 -23544.467} C_VEL
LIN {X 0,Y 228.607,Z 566.849,A -85,B 0,C 180,E1 -23545.226,E2 -23545.226} C_VEL
LIN {X 0,Y 230.93,Z 552.023,A -85,B 0,C 180,E1 -23545.78,E2 -23545.78} C_VEL
LIN {X 0,Y 235.83,Z 495.184,A -85,B 0,C 180,E1 -23547.24,E2 -23547.24} C_VEL
LIN {X 0,Y 231.922,Z 485.697,A -85,B 0,C 180,E1 -23549.731,E2 -23549.731} C_VEL
LIN {X 0,Y 227.549,Z 475.951,A -85,B 0,C 180,E1 -23552.872,E2 -23552.872} C_VEL
LIN {X 0,Y 224.621,Z 470.158,A -85,B 0,C 180,E1 -23555.25,E2 -23555.25} C_VEL
LIN {X 0,Y 222.114,Z 465.403,A -85,B 0,C 180,E1 -23557.563,E2 -23557.563} C_VEL
LIN {X 0,Y 220.82,Z 462.993,A -85,B 0,C 180,E1 -23558.898,E2 -23558.898} C_VEL
LIN {X 0,Y 218.443,Z 459.271,A -85,B 0,C 180,E1 -23561.641,E2 -23561.641} C_VEL
LIN {X 0,Y 216.139,Z 455.816,A -85,B 0,C 180,E1 -23565.027,E2 -23565.027} C_VEL
LIN {X 0,Y 215.704,Z 454.915,A -85,B 0,C 180,E1 -23565.857,E2 -23565.857} C_VEL
LIN {X 0,Y 213.536,Z 451.995,A -85,B 0,C 180,E1 -23571.722,E2 -23571.722} C_VEL
LIN {X 0,Y 213.342,Z 450.402,A -85,B 0,C 180,E1 -23574.329,E2 -23574.329} C_VEL
LIN {X 0,Y 213.415,Z 450.203,A -85,B 0,C 180,E1 -23576.729,E2 -23576.729} C_VEL
LIN {X 0,Y 214.893,Z 454.178,A -85,B 0,C 180,E1 -23583.047,E2 -23583.047} C_VEL
LIN {X 0,Y 216.034,Z 455.152,A -85,B 0,C 180,E1 -23585.163,E2 -23585.163} C_VEL
LIN {X 0,Y 218.065,Z 458.741,A -85,B 0,C 180,E1 -23588.34,E2 -23588.34} C_VEL
LIN {X 0,Y 219.089,Z 460.1,A -85,B 0,C 180,E1 -23589.609,E2 -23589.609} C_VEL
LIN {X 0,Y 221.954,Z 464.592,A -85,B 0,C 180,E1 -23592.691,E2 -23592.691} C_VEL
LIN {X 0,Y 224.646,Z 469.036,A -85,B 0,C 180,E1 -23595.132,E2 -23595.132} C_VEL
LIN {X 0,Y 228.357,Z 475.017,A -85,B 0,C 180,E1 -23598.001,E2 -23598.001} C_VEL
LIN {X 0,Y 233.278,Z 483.763,A -85,B 0,C 180,E1 -23601.282,E2 -23601.282} C_VEL
LIN {X 0,Y 236.247,Z 489.491,A -85,B 0,C 180,E1 -23603.056,E2 -23603.056} C_VEL
LIN {X 0,Y 231.347,Z 545.033,A -85,B 0,C 180,E1 -23604.438,E2 -23604.438} C_VEL
LIN {X 0,Y 228.937,Z 560.899,A -85,B 0,C 180,E1 -23605.095,E2 -23605.095} C_VEL
LIN {X 0,Y 225.868,Z 574.205,A -85,B 0,C 180,E1 -23605.826,E2 -23605.826} C_VEL
LIN {X 0,Y 221.646,Z 588.92,A -85,B 0,C 180,E1 -23606.974,E2 -23606.974} C_VEL
LIN {X 0,Y 217.202,Z 601.073,A -85,B 0,C 180,E1 -23608.148,E2 -23608.148} C_VEL
LIN {X 0,Y 212.15,Z 613.196,A -85,B 0,C 180,E1 -23609.685,E2 -23609.685} C_VEL
LIN {X 0,Y 206.222,Z 625.242,A -85,B 0,C 180,E1 -23611.571,E2 -23611.571} C_VEL
LIN {X 0,Y 199.603,Z 636.825,A -85,B 0,C 180,E1 -23613.848,E2 -23613.848} C_VEL
LIN {X 0,Y 192.587,Z 647.684,A -85,B 0,C 180,E1 -23616.598,E2 -23616.598} C_VEL
LIN {X 0,Y 186.444,Z 656.334,A -85,B 0,C 180,E1 -23619.399,E2 -23619.399} C_VEL
LIN {X 0,Y 179.823,Z 664.749,A -85,B 0,C 180,E1 -23622.878,E2 -23622.878} C_VEL
LIN {X 0,Y 173.662,Z 671.939,A -85,B 0,C 180,E1 -23626.758,E2 -23626.758} C_VEL
LIN {X 0,Y 168.018,Z 678.048,A -85,B 0,C 180,E1 -23631.139,E2 -23631.139} C_VEL
LIN {X 0,Y 163.188,Z 682.919,A -85,B 0,C 180,E1 -23635.953,E2 -23635.953} C_VEL
LIN {X 0,Y 159.483,Z 686.431,A -85,B 0,C 180,E1 -23641.005,E2 -23641.005} C_VEL
LIN {X 0,Y 156.844,Z 688.683,A -85,B 0,C 180,E1 -23646.217,E2 -23646.217} C_VEL
LIN {X 0,Y 155.26,Z 689.755,A -85,B 0,C 180,E1 -23651.918,E2 -23651.918} C_VEL
LIN {X 0,Y 154.545,Z 689.628,A -85,B 0,C 180,E1 -23656.857,E2 -23656.857} C_VEL
LIN {X 0,Y 154.541,Z 688.323,A -85,B 0,C 180,E1 -23662.159,E2 -23662.159} C_VEL
LIN {X 0,Y 155.026,Z 686.721,A -85,B 0,C 180,E1 -23665.852,E2 -23665.852} C_VEL
LIN {X 0,Y 155.536,Z 684.184,A -85,B 0,C 180,E1 -23670,E2 -23670} C_VEL
LIN {X 0,Y 156.921,Z 679.916,A -85,B 0,C 180,E1 -23675.139,E2 -23675.139} C_VEL
LIN {X 0,Y 159.259,Z 674.319,A -85,B 0,C 180,E1 -23680.167,E2 -23680.167} C_VEL
LIN {X 0,Y 162.572,Z 667.236,A -85,B 0,C 180,E1 -23685.033,E2 -23685.033} C_VEL
LIN {X 0,Y 166.238,Z 659.664,A -85,B 0,C 180,E1 -23689.126,E2 -23689.126} C_VEL
LIN {X 0,Y 170.614,Z 650.565,A -85,B 0,C 180,E1 -23693.037,E2 -23693.037} C_VEL
LIN {X 0,Y 174.996,Z 641.292,A -85,B 0,C 180,E1 -23696.217,E2 -23696.217} C_VEL
LIN {X 0,Y 180.194,Z 629.326,A -85,B 0,C 180,E1 -23699.499,E2 -23699.499} C_VEL
LIN {X 0,Y 184.994,Z 617.119,A -85,B 0,C 180,E1 -23702.132,E2 -23702.132} C_VEL
LIN {X 0,Y 189.637,Z 603.691,A -85,B 0,C 180,E1 -23704.414,E2 -23704.414} C_VEL
LIN {X 0,Y 193.525,Z 590.501,A -85,B 0,C 180,E1 -23706.167,E2 -23706.167} C_VEL
LIN {X 0,Y 197.005,Z 576.029,A -85,B 0,C 180,E1 -23707.656,E2 -23707.656} C_VEL
LIN {X 0,Y 199.961,Z 560.224,A -85,B 0,C 180,E1 -23708.841,E2 -23708.841} C_VEL
LIN {X 0,Y 201.921,Z 544.986,A -85,B 0,C 180,E1 -23709.617,E2 -23709.617} C_VEL
LIN {X 0,Y 207.395,Z 467.423,A -85,B 0,C 180,E1 -23711.976,E2 -23711.976} C_VEL
LIN {X 0,Y 201.577,Z 455.531,A -85,B 0,C 180,E1 -23714.478,E2 -23714.478} C_VEL
LIN {X 0,Y 195.285,Z 444.45,A -85,B 0,C 180,E1 -23717.41,E2 -23717.41} C_VEL
LIN {X 0,Y 188.598,Z 433.863,A -85,B 0,C 180,E1 -23720.919,E2 -23720.919} C_VEL
LIN {X 0,Y 182.913,Z 425.762,A -85,B 0,C 180,E1 -23724.337,E2 -23724.337} C_VEL
LIN {X 0,Y 179.551,Z 421.276,A -85,B 0,C 180,E1 -23726.618,E2 -23726.618} C_VEL
LIN {X 0,Y 176.693,Z 417.417,A -85,B 0,C 180,E1 -23728.779,E2 -23728.779} C_VEL
LIN {X 0,Y 173.375,Z 413.602,A -85,B 0,C 180,E1 -23731.555,E2 -23731.555} C_VEL
LIN {X 0,Y 172.359,Z 411.835,A -85,B 0,C 180,E1 -23732.56,E2 -23732.56} C_VEL
LIN {X 0,Y 169.786,Z 409.611,A -85,B 0,C 180,E1 -23735.094,E2 -23735.094} C_VEL
LIN {X 0,Y 168.086,Z 406.444,A -85,B 0,C 180,E1 -23737.246,E2 -23737.246} C_VEL
LIN {X 0,Y 165.42,Z 404.763,A -85,B 0,C 180,E1 -23740.801,E2 -23740.801} C_VEL
LIN {X 0,Y 163.763,Z 402.216,A -85,B 0,C 180,E1 -23743.961,E2 -23743.961} C_VEL
LIN {X 0,Y 163.264,Z 400.605,A -85,B 0,C 180,E1 -23745.35,E2 -23745.35} C_VEL
LIN {X 0,Y 161.188,Z 399.691,A -85,B 0,C 180,E1 -23754.996,E2 -23754.996} C_VEL
LIN {X 0,Y 161.993,Z 399.833,A -85,B 0,C 180,E1 -23760.62,E2 -23760.62} C_VEL
LIN {X 0,Y 163.58,Z 400.722,A -85,B 0,C 180,E1 -23764.928,E2 -23764.928} C_VEL
LIN {X 0,Y 165.04,Z 403.932,A -85,B 0,C 180,E1 -23768.108,E2 -23768.108} C_VEL
LIN {X 0,Y 167.864,Z 406.27,A -85,B 0,C 180,E1 -23772.082,E2 -23772.082} C_VEL
LIN {X 0,Y 168.376,Z 406.95,A -85,B 0,C 180,E1 -23772.734,E2 -23772.734} C_VEL
LIN {X 0,Y 170.219,Z 409.993,A -85,B 0,C 180,E1 -23774.953,E2 -23774.953} C_VEL
LIN {X 0,Y 172.656,Z 412.143,A -85,B 0,C 180,E1 -23777.316,E2 -23777.316} C_VEL
LIN {X 0,Y 174.868,Z 415.517,A -85,B 0,C 180,E1 -23779.363,E2 -23779.363} C_VEL
LIN {X 0,Y 176.781,Z 417.447,A -85,B 0,C 180,E1 -23780.882,E2 -23780.882} C_VEL
LIN {X 0,Y 179.442,Z 421.153,A -85,B 0,C 180,E1 -23782.904,E2 -23782.904} C_VEL
LIN {X 0,Y 180.816,Z 422.842,A -85,B 0,C 180,E1 -23783.857,E2 -23783.857} C_VEL
LIN {X 0,Y 184.375,Z 427.846,A -85,B 0,C 180,E1 -23786.188,E2 -23786.188} C_VEL
LIN {X 0,Y 187.471,Z 432.236,A -85,B 0,C 180,E1 -23788.038,E2 -23788.038} C_VEL
LIN {X 0,Y 192.213,Z 439.516,A -85,B 0,C 180,E1 -23790.637,E2 -23790.637} C_VEL
LIN {X 0,Y 197.322,Z 449.829,A -85,B 0,C 180,E1 -23793.279,E2 -23793.279} C_VEL
LIN {X 0,Y 202.615,Z 462.163,A -85,B 0,C 180,E1 -23795.826,E2 -23795.826} C_VEL
LIN {X 0,Y 206.547,Z 472.419,A -85,B 0,C 180,E1 -23797.613,E2 -23797.613} C_VEL
LIN {X 0,Y 207.086,Z 473.913,A -85,B 0,C 180,E1 -23797.853,E2 -23797.853} C_VEL
LIN {X 0,Y 201.51,Z 553.467,A -85,B 0,C 180,E1 -23800.277,E2 -23800.277} C_VEL
LIN {X 0,Y 199.306,Z 569.671,A -85,B 0,C 180,E1 -23801.085,E2 -23801.085} C_VEL
LIN {X 0,Y 198.878,Z 571.967,A -85,B 0,C 180,E1 -23801.231,E2 -23801.231} C_VEL
LIN {X 0,Y 196.603,Z 579.439,A -85,B 0,C 180,E1 -23801.523,E2 -23801.523} C_VEL
LIN {X 0,Y 189.648,Z 593.697,A -85,B 0,C 180,E1 -23801.789,E2 -23801.789} C_VEL
LIN {X 0,Y 187.382,Z 599.043,A -85,B 0,C 180,E1 -23802.157,E2 -23802.157} C_VEL
LIN {X 0,Y 186.795,Z 600.78,A -85,B 0,C 180,E1 -23802.351,E2 -23802.351} C_VEL
LIN {X 0,Y 182.556,Z 614.144,A -85,B 0,C 180,E1 -23804.191,E2 -23804.191} C_VEL
LIN {X 0,Y 178.466,Z 625.082,A -85,B 0,C 180,E1 -23806.046,E2 -23806.046} C_VEL
LIN {X 0,Y 173.298,Z 637.698,A -85,B 0,C 180,E1 -23808.775,E2 -23808.775} C_VEL
LIN {X 0,Y 167.997,Z 649.138,A -85,B 0,C 180,E1 -23811.899,E2 -23811.899} C_VEL
LIN {X 0,Y 163.273,Z 659.148,A -85,B 0,C 180,E1 -23815.412,E2 -23815.412} C_VEL
LIN {X 0,Y 158.753,Z 668.224,A -85,B 0,C 180,E1 -23819.395,E2 -23819.395} C_VEL
LIN {X 0,Y 154.805,Z 676.062,A -85,B 0,C 180,E1 -23823.727,E2 -23823.727} C_VEL
LIN {X 0,Y 151.75,Z 682.546,A -85,B 0,C 180,E1 -23828.253,E2 -23828.253} C_VEL
LIN {X 0,Y 149.396,Z 688.491,A -85,B 0,C 180,E1 -23833.605,E2 -23833.605} C_VEL
LIN {X 0,Y 148.061,Z 693.029,A -85,B 0,C 180,E1 -23839.055,E2 -23839.055} C_VEL
LIN {X 0,Y 147.637,Z 696.268,A -85,B 0,C 180,E1 -23844.537,E2 -23844.537} C_VEL
LIN {X 0,Y 147.673,Z 697.649,A -85,B 0,C 180,E1 -23848.022,E2 -23848.022} C_VEL
LIN {X 0,Y 147.673,Z 698.618,A -85,B 0,C 180,E1 -23851.978,E2 -23851.978} C_VEL
LIN {X 0,Y 147.566,Z 698.97,A -85,B 0,C 180,E1 -23855.466,E2 -23855.466} C_VEL
LIN {X 0,Y 148.074,Z 698.593,A -85,B 0,C 180,E1 -23860.944,E2 -23860.944} C_VEL
LIN {X 0,Y 149.553,Z 697.105,A -85,B 0,C 180,E1 -23866.377,E2 -23866.377} C_VEL
LIN {X 0,Y 152.243,Z 694.461,A -85,B 0,C 180,E1 -23871.673,E2 -23871.673} C_VEL
LIN {X 0,Y 156.105,Z 690.598,A -85,B 0,C 180,E1 -23876.757,E2 -23876.757} C_VEL
LIN {X 0,Y 161.068,Z 685.467,A -85,B 0,C 180,E1 -23881.574,E2 -23881.574} C_VEL
LIN {X 0,Y 167.273,Z 678.938,A -85,B 0,C 180,E1 -23886.03,E2 -23886.03} C_VEL
LIN {X 0,Y 172.661,Z 672.609,A -85,B 0,C 180,E1 -23889.425,E2 -23889.425} C_VEL
LIN {X 0,Y 180.054,Z 663.58,A -85,B 0,C 180,E1 -23893.084,E2 -23893.084} C_VEL
LIN {X 0,Y 187.508,Z 653.535,A -85,B 0,C 180,E1 -23896.179,E2 -23896.179} C_VEL
LIN {X 0,Y 194.324,Z 643.313,A -85,B 0,C 180,E1 -23898.63,E2 -23898.63} C_VEL
LIN {X 0,Y 201.361,Z 631.405,A -85,B 0,C 180,E1 -23900.844,E2 -23900.844} C_VEL
LIN {X 0,Y 205.712,Z 622.774,A -85,B 0,C 180,E1 -23902.19,E2 -23902.19} C_VEL
LIN {X 0,Y 211.507,Z 610.346,A -85,B 0,C 180,E1 -23903.686,E2 -23903.686} C_VEL
LIN {X 0,Y 216.688,Z 596.917,A -85,B 0,C 180,E1 -23904.98,E2 -23904.98} C_VEL
LIN {X 0,Y 221.404,Z 582.01,A -85,B 0,C 180,E1 -23906.025,E2 -23906.025} C_VEL
LIN {X 0,Y 225.007,Z 567.138,A -85,B 0,C 180,E1 -23906.773,E2 -23906.773} C_VEL
LIN {X 0,Y 227.481,Z 551.979,A -85,B 0,C 180,E1 -23907.329,E2 -23907.329} C_VEL
LIN {X 0,Y 232.28,Z 498.393,A -85,B 0,C 180,E1 -23908.685,E2 -23908.685} C_VEL
LIN {X 0,Y 228.208,Z 488.309,A -85,B 0,C 180,E1 -23911.522,E2 -23911.522} C_VEL
LIN {X 0,Y 224.392,Z 479.741,A -85,B 0,C 180,E1 -23914.548,E2 -23914.548} C_VEL
LIN {X 0,Y 221.562,Z 473.935,A -85,B 0,C 180,E1 -23917.127,E2 -23917.127} C_VEL
LIN {X 0,Y 219.316,Z 469.563,A -85,B 0,C 180,E1 -23919.483,E2 -23919.483} C_VEL
LIN {X 0,Y 217.165,Z 466.051,A -85,B 0,C 180,E1 -23922.096,E2 -23922.096} C_VEL
LIN {X 0,Y 214.957,Z 462.528,A -85,B 0,C 180,E1 -23925.532,E2 -23925.532} C_VEL
LIN {X 0,Y 214.591,Z 461.788,A -85,B 0,C 180,E1 -23926.265,E2 -23926.265} C_VEL
LIN {X 0,Y 212.627,Z 459.061,A -85,B 0,C 180,E1 -23931.873,E2 -23931.873} C_VEL
LIN {X 0,Y 212.459,Z 457.365,A -85,B 0,C 180,E1 -23934.782,E2 -23934.782} C_VEL
LIN {X 0,Y 212.541,Z 457.263,A -85,B 0,C 180,E1 -23936.715,E2 -23936.715} C_VEL
LIN {X 0,Y 213.778,Z 461.023,A -85,B 0,C 180,E1 -23942.533,E2 -23942.533} C_VEL
LIN {X 0,Y 214.938,Z 462.174,A -85,B 0,C 180,E1 -23944.837,E2 -23944.837} C_VEL
LIN {X 0,Y 217.069,Z 465.831,A -85,B 0,C 180,E1 -23948.232,E2 -23948.232} C_VEL
LIN {X 0,Y 217.882,Z 467.059,A -85,B 0,C 180,E1 -23949.282,E2 -23949.282} C_VEL
LIN {X 0,Y 220.375,Z 471.086,A -85,B 0,C 180,E1 -23952.081,E2 -23952.081} C_VEL
LIN {X 0,Y 223.118,Z 475.831,A -85,B 0,C 180,E1 -23954.684,E2 -23954.684} C_VEL
LIN {X 0,Y 226.319,Z 481.204,A -85,B 0,C 180,E1 -23957.275,E2 -23957.275} C_VEL
LIN {X 0,Y 230.66,Z 489.237,A -85,B 0,C 180,E1 -23960.338,E2 -23960.338} C_VEL
LIN {X 0,Y 232.647,Z 493.097,A -85,B 0,C 180,E1 -23961.604,E2 -23961.604} C_VEL
LIN {X 0,Y 227.902,Z 545.156,A -85,B 0,C 180,E1 -23962.886,E2 -23962.886} C_VEL
LIN {X 0,Y 225.428,Z 561.072,A -85,B 0,C 180,E1 -23963.541,E2 -23963.541} C_VEL
LIN {X 0,Y 222.176,Z 574.783,A -85,B 0,C 180,E1 -23964.283,E2 -23964.283} C_VEL
LIN {X 0,Y 217.863,Z 589.315,A -85,B 0,C 180,E1 -23965.412,E2 -23965.412} C_VEL
LIN {X 0,Y 213.198,Z 601.667,A -85,B 0,C 180,E1 -23966.598,E2 -23966.598} C_VEL
LIN {X 0,Y 207.484,Z 614.773,A -85,B 0,C 180,E1 -23968.275,E2 -23968.275} C_VEL
LIN {X 0,Y 201.251,Z 626.798,A -85,B 0,C 180,E1 -23970.196,E2 -23970.196} C_VEL
LIN {X 0,Y 194.021,Z 638.792,A -85,B 0,C 180,E1 -23972.629,E2 -23972.629} C_VEL
LIN {X 0,Y 187.176,Z 648.827,A -85,B 0,C 180,E1 -23975.248,E2 -23975.248} C_VEL
LIN {X 0,Y 179.796,Z 658.593,A -85,B 0,C 180,E1 -23978.577,E2 -23978.577} C_VEL
LIN {X 0,Y 172.995,Z 666.665,A -85,B 0,C 180,E1 -23982.148,E2 -23982.148} C_VEL
LIN {X 0,Y 166.557,Z 673.709,A -85,B 0,C 180,E1 -23986.27,E2 -23986.27} C_VEL
LIN {X 0,Y 160.919,Z 679.384,A -85,B 0,C 180,E1 -23990.708,E2 -23990.708} C_VEL
LIN {X 0,Y 157.126,Z 682.93,A -85,B 0,C 180,E1 -23994.446,E2 -23994.446} C_VEL
LIN {X 0,Y 153.059,Z 686.51,A -85,B 0,C 180,E1 -23999.663,E2 -23999.663} C_VEL
LIN {X 0,Y 150.155,Z 688.828,A -85,B 0,C 180,E1 -24005.087,E2 -24005.087} C_VEL
LIN {X 0,Y 148.4,Z 689.945,A -85,B 0,C 180,E1 -24010.64,E2 -24010.64} C_VEL
LIN {X 0,Y 147.512,Z 689.88,A -85,B 0,C 180,E1 -24016.219,E2 -24016.219} C_VEL
LIN {X 0,Y 147.415,Z 688.624,A -85,B 0,C 180,E1 -24021.777,E2 -24021.777} C_VEL
LIN {X 0,Y 147.948,Z 686.887,A -85,B 0,C 180,E1 -24026.023,E2 -24026.023} C_VEL
LIN {X 0,Y 148.426,Z 684.58,A -85,B 0,C 180,E1 -24030,E2 -24030} C_VEL
LIN {X 0,Y 149.85,Z 680.38,A -85,B 0,C 180,E1 -24035.382,E2 -24035.382} C_VEL
LIN {X 0,Y 152.305,Z 674.854,A -85,B 0,C 180,E1 -24040.637,E2 -24040.637} C_VEL
LIN {X 0,Y 155.745,Z 667.851,A -85,B 0,C 180,E1 -24045.709,E2 -24045.709} C_VEL
LIN {X 0,Y 159.585,Z 660.366,A -85,B 0,C 180,E1 -24049.957,E2 -24049.957} C_VEL
LIN {X 0,Y 164.144,Z 651.36,A -85,B 0,C 180,E1 -24054.001,E2 -24054.001} C_VEL
LIN {X 0,Y 169.469,Z 640.486,A -85,B 0,C 180,E1 -24057.811,E2 -24057.811} C_VEL
LIN {X 0,Y 174.527,Z 629.322,A -85,B 0,C 180,E1 -24060.893,E2 -24060.893} C_VEL
LIN {X 0,Y 179.547,Z 617.068,A -85,B 0,C 180,E1 -24063.566,E2 -24063.566} C_VEL
LIN {X 0,Y 184.383,Z 603.568,A -85,B 0,C 180,E1 -24065.877,E2 -24065.877} C_VEL
LIN {X 0,Y 188.418,Z 590.323,A -85,B 0,C 180,E1 -24067.647,E2 -24067.647} C_VEL
LIN {X 0,Y 192.01,Z 575.746,A -85,B 0,C 180,E1 -24069.153,E2 -24069.153} C_VEL
LIN {X 0,Y 194.949,Z 560.527,A -85,B 0,C 180,E1 -24070.29,E2 -24070.29} C_VEL
LIN {X 0,Y 197.008,Z 545.035,A -85,B 0,C 180,E1 -24071.085,E2 -24071.085} C_VEL
LIN {X 0,Y 202.539,Z 470.12,A -85,B 0,C 180,E1 -24073.367,E2 -24073.367} C_VEL
LIN {X 0,Y 196.632,Z 458.064,A -85,B 0,C 180,E1 -24076.092,E2 -24076.092} C_VEL
LIN {X 0,Y 191.506,Z 448.969,A -85,B 0,C 180,E1 -24078.655,E2 -24078.655} C_VEL
LIN {X 0,Y 185.412,Z 439.138,A -85,B 0,C 180,E1 -24082.062,E2 -24082.062} C_VEL
LIN {X 0,Y 180.298,Z 431.616,A -85,B 0,C 180,E1 -24085.328,E2 -24085.328} C_VEL
LIN {X 0,Y 176.941,Z 427.076,A -85,B 0,C 180,E1 -24087.741,E2 -24087.741} C_VEL
LIN {X 0,Y 174.082,Z 423.145,A -85,B 0,C 180,E1 -24090.055,E2 -24090.055} C_VEL
LIN {X 0,Y 171.317,Z 419.694,A -85,B 0,C 180,E1 -24092.555,E2 -24092.555} C_VEL
LIN {X 0,Y 170.525,Z 418.415,A -85,B 0,C 180,E1 -24093.37,E2 -24093.37} C_VEL
LIN {X 0,Y 168.063,Z 416.028,A -85,B 0,C 180,E1 -24095.963,E2 -24095.963} C_VEL
LIN {X 0,Y 166.584,Z 413.284,A -85,B 0,C 180,E1 -24097.94,E2 -24097.94} C_VEL
LIN {X 0,Y 164.009,Z 411.396,A -85,B 0,C 180,E1 -24101.626,E2 -24101.626} C_VEL
LIN {X 0,Y 162.507,Z 408.762,A -85,B 0,C 180,E1 -24104.799,E2 -24104.799} C_VEL
LIN {X 0,Y 162.145,Z 407.599,A -85,B 0,C 180,E1 -24105.887,E2 -24105.887} C_VEL
LIN {X 0,Y 160.318,Z 406.736,A -85,B 0,C 180,E1 -24114.969,E2 -24114.969} C_VEL
LIN {X 0,Y 161.097,Z 406.879,A -85,B 0,C 180,E1 -24120.545,E2 -24120.545} C_VEL
LIN {X 0,Y 162.424,Z 407.654,A -85,B 0,C 180,E1 -24124.342,E2 -24124.342} C_VEL
LIN {X 0,Y 163.979,Z 410.959,A -85,B 0,C 180,E1 -24127.851,E2 -24127.851} C_VEL
LIN {X 0,Y 166.791,Z 413.494,A -85,B 0,C 180,E1 -24131.926,E2 -24131.926} C_VEL
LIN {X 0,Y 168.616,Z 416.589,A -85,B 0,C 180,E1 -24134.25,E2 -24134.25} C_VEL
LIN {X 0,Y 170.917,Z 418.835,A -85,B 0,C 180,E1 -24136.612,E2 -24136.612} C_VEL
LIN {X 0,Y 173.505,Z 422.553,A -85,B 0,C 180,E1 -24139.06,E2 -24139.06} C_VEL
LIN {X 0,Y 174.843,Z 424.074,A -85,B 0,C 180,E1 -24140.174,E2 -24140.174} C_VEL
LIN {X 0,Y 178.71,Z 429.379,A -85,B 0,C 180,E1 -24143.157,E2 -24143.157} C_VEL
LIN {X 0,Y 182.429,Z 434.689,A -85,B 0,C 180,E1 -24145.683,E2 -24145.683} C_VEL
LIN {X 0,Y 187.751,Z 442.695,A -85,B 0,C 180,E1 -24148.888,E2 -24148.888} C_VEL
LIN {X 0,Y 190.972,Z 448.774,A -85,B 0,C 180,E1 -24150.704,E2 -24150.704} C_VEL
LIN {X 0,Y 196.112,Z 460.214,A -85,B 0,C 180,E1 -24153.434,E2 -24153.434} C_VEL
LIN {X 0,Y 201.212,Z 473.29,A -85,B 0,C 180,E1 -24155.96,E2 -24155.96} C_VEL
LIN {X 0,Y 202.225,Z 476.247,A -85,B 0,C 180,E1 -24156.451,E2 -24156.451} C_VEL
LIN {X 0,Y 196.516,Z 553.86,A -85,B 0,C 180,E1 -24158.834,E2 -24158.834} C_VEL
LIN {X 0,Y 194.228,Z 569.839,A -85,B 0,C 180,E1 -24159.642,E2 -24159.642} C_VEL
LIN {X 0,Y 191.192,Z 584.471,A -85,B 0,C 180,E1 -24160.698,E2 -24160.698} C_VEL
LIN {X 0,Y 187.426,Z 598.602,A -85,B 0,C 180,E1 -24162.079,E2 -24162.079} C_VEL
LIN {X 0,Y 186.795,Z 600.78,A -85,B 0,C 180,E1 -24162.351,E2 -24162.351} C_VEL
LIN {X 0,Y 184.687,Z 606.085,A -85,B 0,C 180,E1 -24162.875,E2 -24162.875} C_VEL
LIN {X 0,Y 179.696,Z 614.408,A -85,B 0,C 180,E1 -24163.476,E2 -24163.476} C_VEL
LIN {X 0,Y 174.497,Z 622.498,A -85,B 0,C 180,E1 -24164.24,E2 -24164.24} C_VEL
LIN {X 0,Y 172.061,Z 627.286,A -85,B 0,C 180,E1 -24165.042,E2 -24165.042} C_VEL
LIN {X 0,Y 166.993,Z 638.876,A -85,B 0,C 180,E1 -24167.672,E2 -24167.672} C_VEL
LIN {X 0,Y 161.546,Z 650.102,A -85,B 0,C 180,E1 -24170.889,E2 -24170.889} C_VEL
LIN {X 0,Y 156.827,Z 659.594,A -85,B 0,C 180,E1 -24174.368,E2 -24174.368} C_VEL
LIN {X 0,Y 151.945,Z 668.868,A -85,B 0,C 180,E1 -24178.644,E2 -24178.644} C_VEL
LIN {X 0,Y 147.878,Z 676.553,A -85,B 0,C 180,E1 -24183.16,E2 -24183.16} C_VEL
LIN {X 0,Y 144.35,Z 683.718,A -85,B 0,C 180,E1 -24188.583,E2 -24188.583} C_VEL
LIN {X 0,Y 142.053,Z 689.344,A -85,B 0,C 180,E1 -24194.21,E2 -24194.21} C_VEL
LIN {X 0,Y 141.053,Z 692.672,A -85,B 0,C 180,E1 -24198.504,E2 -24198.504} C_VEL
LIN {X 0,Y 140.543,Z 695.948,A -85,B 0,C 180,E1 -24204.26,E2 -24204.26} C_VEL
LIN {X 0,Y 140.601,Z 697.549,A -85,B 0,C 180,E1 -24208.569,E2 -24208.569} C_VEL
LIN {X 0,Y 140.593,Z 698.237,A -85,B 0,C 180,E1 -24211.289,E2 -24211.289} C_VEL
LIN {X 0,Y 140.494,Z 698.739,A -85,B 0,C 180,E1 -24215.742,E2 -24215.742} C_VEL
LIN {X 0,Y 141.069,Z 698.409,A -85,B 0,C 180,E1 -24221.495,E2 -24221.495} C_VEL
LIN {X 0,Y 142.715,Z 696.972,A -85,B 0,C 180,E1 -24227.186,E2 -24227.186} C_VEL
LIN {X 0,Y 145.592,Z 694.354,A -85,B 0,C 180,E1 -24232.717,E2 -24232.717} C_VEL
LIN {X 0,Y 149.733,Z 690.544,A -85,B 0,C 180,E1 -24237.993,E2 -24237.993} C_VEL
LIN {X 0,Y 155.007,Z 685.469,A -85,B 0,C 180,E1 -24242.962,E2 -24242.962} C_VEL
LIN {X 0,Y 161.549,Z 679.001,A -85,B 0,C 180,E1 -24247.521,E2 -24247.521} C_VEL
LIN {X 0,Y 167.875,Z 671.968,A -85,B 0,C 180,E1 -24251.331,E2 -24251.331} C_VEL
LIN {X 0,Y 174.92,Z 663.784,A -85,B 0,C 180,E1 -24254.678,E2 -24254.678} C_VEL
LIN {X 0,Y 182.662,Z 653.828,A -85,B 0,C 180,E1 -24257.787,E2 -24257.787} C_VEL
LIN {X 0,Y 189.723,Z 643.67,A -85,B 0,C 180,E1 -24260.233,E2 -24260.233} C_VEL
LIN {X 0,Y 196.871,Z 632.046,A -85,B 0,C 180,E1 -24262.41,E2 -24262.41} C_VEL
LIN {X 0,Y 201.458,Z 623.376,A -85,B 0,C 180,E1 -24263.778,E2 -24263.778} C_VEL
LIN {X 0,Y 207.42,Z 611.128,A -85,B 0,C 180,E1 -24265.252,E2 -24265.252} C_VEL
LIN {X 0,Y 212.726,Z 597.899,A -85,B 0,C 180,E1 -24266.533,E2 -24266.533} C_VEL
LIN {X 0,Y 217.569,Z 583.35,A -85,B 0,C 180,E1 -24267.554,E2 -24267.554} C_VEL
LIN {X 0,Y 221.384,Z 568.24,A -85,B 0,C 180,E1 -24268.341,E2 -24268.341} C_VEL
LIN {X 0,Y 224.109,Z 552.621,A -85,B 0,C 180,E1 -24268.904,E2 -24268.904} C_VEL
LIN {X 0,Y 228.829,Z 501.576,A -85,B 0,C 180,E1 -24270.204,E2 -24270.204} C_VEL
LIN {X 0,Y 225.199,Z 492.378,A -85,B 0,C 180,E1 -24272.963,E2 -24272.963} C_VEL
LIN {X 0,Y 221.749,Z 484.173,A -85,B 0,C 180,E1 -24275.982,E2 -24275.982} C_VEL
LIN {X 0,Y 218.066,Z 476.441,A -85,B 0,C 180,E1 -24279.822,E2 -24279.822} C_VEL
LIN {X 0,Y 215.785,Z 472.694,A -85,B 0,C 180,E1 -24282.712,E2 -24282.712} C_VEL
LIN {X 0,Y 213.659,Z 468.945,A -85,B 0,C 180,E1 -24286.325,E2 -24286.325} C_VEL
LIN {X 0,Y 211.625,Z 465.496,A -85,B 0,C 180,E1 -24292.971,E2 -24292.971} C_VEL
LIN {X 0,Y 211.591,Z 464.328,A -85,B 0,C 180,E1 -24295.174,E2 -24295.174} C_VEL
LIN {X 0,Y 211.674,Z 464.428,A -85,B 0,C 180,E1 -24296.877,E2 -24296.877} C_VEL
LIN {X 0,Y 212.512,Z 467.594,A -85,B 0,C 180,E1 -24301.541,E2 -24301.541} C_VEL
LIN {X 0,Y 213.814,Z 469.035,A -85,B 0,C 180,E1 -24304.419,E2 -24304.419} C_VEL
LIN {X 0,Y 215.965,Z 472.785,A -85,B 0,C 180,E1 -24307.98,E2 -24307.98} C_VEL
LIN {X 0,Y 218.741,Z 477.468,A -85,B 0,C 180,E1 -24311.38,E2 -24311.38} C_VEL
LIN {X 0,Y 221.055,Z 481.649,A -85,B 0,C 180,E1 -24313.723,E2 -24313.723} C_VEL
LIN {X 0,Y 224.346,Z 487.404,A -85,B 0,C 180,E1 -24316.552,E2 -24316.552} C_VEL
LIN {X 0,Y 228.524,Z 495.489,A -85,B 0,C 180,E1 -24319.657,E2 -24319.657} C_VEL
LIN {X 0,Y 229.202,Z 496.89,A -85,B 0,C 180,E1 -24320.122,E2 -24320.122} C_VEL
LIN {X 0,Y 224.608,Z 545.609,A -85,B 0,C 180,E1 -24321.305,E2 -24321.305} C_VEL
LIN {X 0,Y 222.049,Z 561.469,A -85,B 0,C 180,E1 -24321.951,E2 -24321.951} C_VEL
LIN {X 0,Y 218.68,Z 575.267,A -85,B 0,C 180,E1 -24322.686,E2 -24322.686} C_VEL
LIN {X 0,Y 214.151,Z 590.017,A -85,B 0,C 180,E1 -24323.823,E2 -24323.823} C_VEL
LIN {X 0,Y 209.355,Z 602.269,A -85,B 0,C 180,E1 -24324.989,E2 -24324.989} C_VEL
LIN {X 0,Y 204.104,Z 613.977,A -85,B 0,C 180,E1 -24326.457,E2 -24326.457} C_VEL
LIN {X 0,Y 197.674,Z 626.183,A -85,B 0,C 180,E1 -24328.364,E2 -24328.364} C_VEL
LIN {X 0,Y 191.408,Z 636.494,A -85,B 0,C 180,E1 -24330.361,E2 -24330.361} C_VEL
LIN {X 0,Y 184.219,Z 646.926,A -85,B 0,C 180,E1 -24332.933,E2 -24332.933} C_VEL
LIN {X 0,Y 176.368,Z 657.066,A -85,B 0,C 180,E1 -24336.203,E2 -24336.203} C_VEL
LIN {X 0,Y 169.11,Z 665.436,A -85,B 0,C 180,E1 -24339.75,E2 -24339.75} C_VEL
LIN {X 0,Y 162.07,Z 672.845,A -85,B 0,C 180,E1 -24343.935,E2 -24343.935} C_VEL
LIN {X 0,Y 155.263,Z 679.357,A -85,B 0,C 180,E1 -24348.978,E2 -24348.978} C_VEL
LIN {X 0,Y 151.17,Z 682.943,A -85,B 0,C 180,E1 -24352.816,E2 -24352.816} C_VEL
LIN {X 0,Y 146.723,Z 686.591,A -85,B 0,C 180,E1 -24358.204,E2 -24358.204} C_VEL
LIN {X 0,Y 143.516,Z 688.973,A -85,B 0,C 180,E1 -24363.85,E2 -24363.85} C_VEL
LIN {X 0,Y 141.501,Z 690.154,A -85,B 0,C 180,E1 -24369.655,E2 -24369.655} C_VEL
LIN {X 0,Y 140.472,Z 690.119,A -85,B 0,C 180,E1 -24375.513,E2 -24375.513} C_VEL
LIN {X 0,Y 140.286,Z 688.925,A -85,B 0,C 180,E1 -24381.356,E2 -24381.356} C_VEL
LIN {X 0,Y 140.916,Z 686.579,A -85,B 0,C 180,E1 -24387.141,E2 -24387.141} C_VEL
LIN {X 0,Y 141.91,Z 683.067,A -85,B 0,C 180,E1 -24392.839,E2 -24392.839} C_VEL
LIN {X 0,Y 144,Z 678.282,A -85,B 0,C 180,E1 -24398.42,E2 -24398.42} C_VEL
LIN {X 0,Y 147,Z 672.121,A -85,B 0,C 180,E1 -24403.831,E2 -24403.831} C_VEL
LIN {X 0,Y 151.183,Z 664.374,A -85,B 0,C 180,E1 -24408.99,E2 -24408.99} C_VEL
LIN {X 0,Y 155.602,Z 656.14,A -85,B 0,C 180,E1 -24413.279,E2 -24413.279} C_VEL
LIN {X 0,Y 160.793,Z 646.227,A -85,B 0,C 180,E1 -24417.319,E2 -24417.319} C_VEL
LIN {X 0,Y 165.875,Z 636.078,A -85,B 0,C 180,E1 -24420.56,E2 -24420.56} C_VEL
LIN {X 0,Y 171.308,Z 623.999,A -85,B 0,C 180,E1 -24423.631,E2 -24423.631} C_VEL
LIN {X 0,Y 176.714,Z 610.57,A -85,B 0,C 180,E1 -24426.27,E2 -24426.27} C_VEL
LIN {X 0,Y 181.346,Z 597.137,A -85,B 0,C 180,E1 -24428.322,E2 -24428.322} C_VEL
LIN {X 0,Y 185.303,Z 583.245,A -85,B 0,C 180,E1 -24429.971,E2 -24429.971} C_VEL
LIN {X 0,Y 188.57,Z 568.984,A -85,B 0,C 180,E1 -24431.24,E2 -24431.24} C_VEL
LIN {X 0,Y 191.144,Z 553.694,A -85,B 0,C 180,E1 -24432.232,E2 -24432.232} C_VEL
LIN {X 0,Y 192.862,Z 538.049,A -85,B 0,C 180,E1 -24432.878,E2 -24432.878} C_VEL
LIN {X 0,Y 197.74,Z 472.746,A -85,B 0,C 180,E1 -24434.852,E2 -24434.852} C_VEL
LIN {X 0,Y 192.642,Z 462.233,A -85,B 0,C 180,E1 -24437.369,E2 -24437.369} C_VEL
LIN {X 0,Y 187.672,Z 453.249,A -85,B 0,C 180,E1 -24440.031,E2 -24440.031} C_VEL
LIN {X 0,Y 182.205,Z 444.222,A -85,B 0,C 180,E1 -24443.307,E2 -24443.307} C_VEL
LIN {X 0,Y 177.554,Z 437.251,A -85,B 0,C 180,E1 -24446.474,E2 -24446.474} C_VEL
LIN {X 0,Y 174.773,Z 433.288,A -85,B 0,C 180,E1 -24448.604,E2 -24448.604} C_VEL
LIN {X 0,Y 172.001,Z 429.422,A -85,B 0,C 180,E1 -24450.972,E2 -24450.972} C_VEL
LIN {X 0,Y 169.245,Z 425.653,A -85,B 0,C 180,E1 -24453.652,E2 -24453.652} C_VEL
LIN {X 0,Y 168.213,Z 424.568,A -85,B 0,C 180,E1 -24454.725,E2 -24454.725} C_VEL
LIN {X 0,Y 165.891,Z 421.615,A -85,B 0,C 180,E1 -24457.506,E2 -24457.506} C_VEL
LIN {X 0,Y 165.175,Z 420.111,A -85,B 0,C 180,E1 -24458.566,E2 -24458.566} C_VEL
LIN {X 0,Y 162.551,Z 417.902,A -85,B 0,C 180,E1 -24462.625,E2 -24462.625} C_VEL
LIN {X 0,Y 161.23,Z 415.196,A -85,B 0,C 180,E1 -24465.806,E2 -24465.806} C_VEL
LIN {X 0,Y 161.041,Z 414.582,A -85,B 0,C 180,E1 -24466.432,E2 -24466.432} C_VEL
LIN {X 0,Y 159.448,Z 413.783,A -85,B 0,C 180,E1 -24474.941,E2 -24474.941} C_VEL
LIN {X 0,Y 160.224,Z 413.919,A -85,B 0,C 180,E1 -24480.548,E2 -24480.548} C_VEL
LIN {X 0,Y 161.341,Z 414.708,A -85,B 0,C 180,E1 -24483.906,E2 -24483.906} C_VEL
LIN {X 0,Y 162.839,Z 417.874,A -85,B 0,C 180,E1 -24487.438,E2 -24487.438} C_VEL
LIN {X 0,Y 165.311,Z 420.247,A -85,B 0,C 180,E1 -24491.22,E2 -24491.22} C_VEL
LIN {X 0,Y 167.532,Z 423.802,A -85,B 0,C 180,E1 -24494.112,E2 -24494.112} C_VEL
LIN {X 0,Y 169.258,Z 425.574,A -85,B 0,C 180,E1 -24495.947,E2 -24495.947} C_VEL
LIN {X 0,Y 171.797,Z 429.186,A -85,B 0,C 180,E1 -24498.445,E2 -24498.445} C_VEL
LIN {X 0,Y 172.923,Z 430.607,A -85,B 0,C 180,E1 -24499.435,E2 -24499.435} C_VEL
LIN {X 0,Y 176.597,Z 435.774,A -85,B 0,C 180,E1 -24502.406,E2 -24502.406} C_VEL
LIN {X 0,Y 181.118,Z 442.41,A -85,B 0,C 180,E1 -24505.574,E2 -24505.574} C_VEL
LIN {X 0,Y 185.762,Z 449.958,A -85,B 0,C 180,E1 -24508.463,E2 -24508.463} C_VEL
LIN {X 0,Y 190.308,Z 459.855,A -85,B 0,C 180,E1 -24511.131,E2 -24511.131} C_VEL
LIN {X 0,Y 195.453,Z 472.758,A -85,B 0,C 180,E1 -24513.92,E2 -24513.92} C_VEL
LIN {X 0,Y 197.463,Z 478.489,A -85,B 0,C 180,E1 -24514.968,E2 -24514.968} C_VEL
LIN {X 0,Y 191.786,Z 553.02,A -85,B 0,C 180,E1 -24517.261,E2 -24517.261} C_VEL
LIN {X 0,Y 189.575,Z 568.434,A -85,B 0,C 180,E1 -24518.02,E2 -24518.02} C_VEL
LIN {X 0,Y 186.307,Z 583.967,A -85,B 0,C 180,E1 -24519.133,E2 -24519.133} C_VEL
LIN {X 0,Y 182.504,Z 597.867,A -85,B 0,C 180,E1 -24520.488,E2 -24520.488} C_VEL
LIN {X 0,Y 178.01,Z 611.916,A -85,B 0,C 180,E1 -24522.353,E2 -24522.353} C_VEL
LIN {X 0,Y 173.365,Z 624.044,A -85,B 0,C 180,E1 -24524.398,E2 -24524.398} C_VEL
LIN {X 0,Y 172.061,Z 627.286,A -85,B 0,C 180,E1 -24525.042,E2 -24525.042} C_VEL
LIN {X 0,Y 169.571,Z 632.021,A -85,B 0,C 180,E1 -24525.903,E2 -24525.903} C_VEL
LIN {X 0,Y 159.135,Z 645.066,A -85,B 0,C 180,E1 -24528.113,E2 -24528.113} C_VEL
LIN {X 0,Y 156.159,Z 649.231,A -85,B 0,C 180,E1 -24529.194,E2 -24529.194} C_VEL
LIN {X 0,Y 155.387,Z 650.567,A -85,B 0,C 180,E1 -24529.638,E2 -24529.638} C_VEL
LIN {X 0,Y 150.234,Z 660.351,A -85,B 0,C 180,E1 -24533.384,E2 -24533.384} C_VEL
LIN {X 0,Y 145.142,Z 669.471,A -85,B 0,C 180,E1 -24537.816,E2 -24537.816} C_VEL
LIN {X 0,Y 140.438,Z 677.992,A -85,B 0,C 180,E1 -24543.231,E2 -24543.231} C_VEL
LIN {X 0,Y 136.929,Z 684.815,A -85,B 0,C 180,E1 -24548.944,E2 -24548.944} C_VEL
LIN {X 0,Y 134.671,Z 690.151,A -85,B 0,C 180,E1 -24554.874,E2 -24554.874} C_VEL
LIN {X 0,Y 133.602,Z 694.126,A -85,B 0,C 180,E1 -24560.92,E2 -24560.92} C_VEL
LIN {X 0,Y 133.479,Z 696.792,A -85,B 0,C 180,E1 -24566.982,E2 -24566.982} C_VEL
LIN {X 0,Y 133.539,Z 697.838,A -85,B 0,C 180,E1 -24570.678,E2 -24570.678} C_VEL
LIN {X 0,Y 133.411,Z 698.507,A -85,B 0,C 180,E1 -24576.048,E2 -24576.048} C_VEL
LIN {X 0,Y 134.069,Z 698.226,A -85,B 0,C 180,E1 -24582.104,E2 -24582.104} C_VEL
LIN {X 0,Y 135.882,Z 696.83,A -85,B 0,C 180,E1 -24588.079,E2 -24588.079} C_VEL
LIN {X 0,Y 139,Z 694.246,A -85,B 0,C 180,E1 -24593.859,E2 -24593.859} C_VEL
LIN {X 0,Y 143.463,Z 690.49,A -85,B 0,C 180,E1 -24599.333,E2 -24599.333} C_VEL
LIN {X 0,Y 149.051,Z 685.472,A -85,B 0,C 180,E1 -24604.459,E2 -24604.459} C_VEL
LIN {X 0,Y 155.918,Z 679.066,A -85,B 0,C 180,E1 -24609.127,E2 -24609.127} C_VEL
LIN {X 0,Y 162.384,Z 672.325,A -85,B 0,C 180,E1 -24612.889,E2 -24612.889} C_VEL
LIN {X 0,Y 169.946,Z 663.988,A -85,B 0,C 180,E1 -24616.361,E2 -24616.361} C_VEL
LIN {X 0,Y 177.971,Z 654.112,A -85,B 0,C 180,E1 -24619.48,E2 -24619.48} C_VEL
LIN {X 0,Y 185.281,Z 644.017,A -85,B 0,C 180,E1 -24621.914,E2 -24621.914} C_VEL
LIN {X 0,Y 192.54,Z 632.664,A -85,B 0,C 180,E1 -24624.051,E2 -24624.051} C_VEL
LIN {X 0,Y 197.366,Z 623.978,A -85,B 0,C 180,E1 -24625.433,E2 -24625.433} C_VEL
LIN {X 0,Y 204.173,Z 610.344,A -85,B 0,C 180,E1 -24627.038,E2 -24627.038} C_VEL
LIN {X 0,Y 208.926,Z 598.799,A -85,B 0,C 180,E1 -24628.144,E2 -24628.144} C_VEL
LIN {X 0,Y 213.873,Z 584.562,A -85,B 0,C 180,E1 -24629.147,E2 -24629.147} C_VEL
LIN {X 0,Y 217.775,Z 569.951,A -85,B 0,C 180,E1 -24629.916,E2 -24629.916} C_VEL
LIN {X 0,Y 220.675,Z 554.762,A -85,B 0,C 180,E1 -24630.467,E2 -24630.467} C_VEL
LIN {X 0,Y 223.068,Z 532.521,A -85,B 0,C 180,E1 -24631.042,E2 -24631.042} C_VEL
LIN {X 0,Y 225.595,Z 505.03,A -85,B 0,C 180,E1 -24631.722,E2 -24631.722} C_VEL
LIN {X 0,Y 222.324,Z 496.382,A -85,B 0,C 180,E1 -24634.461,E2 -24634.461} C_VEL
LIN {X 0,Y 219.443,Z 489.387,A -85,B 0,C 180,E1 -24637.213,E2 -24637.213} C_VEL
LIN {X 0,Y 216.429,Z 482.8,A -85,B 0,C 180,E1 -24640.616,E2 -24640.616} C_VEL
LIN {X 0,Y 214.497,Z 479.414,A -85,B 0,C 180,E1 -24643.241,E2 -24643.241} C_VEL
LIN {X 0,Y 212.389,Z 475.606,A -85,B 0,C 180,E1 -24647.094,E2 -24647.094} C_VEL
LIN {X 0,Y 210.739,Z 472.621,A -85,B 0,C 180,E1 -24653.008,E2 -24653.008} C_VEL
LIN {X 0,Y 210.72,Z 471.377,A -85,B 0,C 180,E1 -24655.211,E2 -24655.211} C_VEL
LIN {X 0,Y 210.784,Z 471.468,A -85,B 0,C 180,E1 -24656.688,E2 -24656.688} C_VEL
LIN {X 0,Y 211.513,Z 474.502,A -85,B 0,C 180,E1 -24661.191,E2 -24661.191} C_VEL
LIN {X 0,Y 212.72,Z 475.896,A -85,B 0,C 180,E1 -24664.027,E2 -24664.027} C_VEL
LIN {X 0,Y 214.72,Z 479.572,A -85,B 0,C 180,E1 -24667.524,E2 -24667.524} C_VEL
LIN {X 0,Y 217.189,Z 483.938,A -85,B 0,C 180,E1 -24670.724,E2 -24670.724} C_VEL
LIN {X 0,Y 220.678,Z 490.336,A -85,B 0,C 180,E1 -24674.29,E2 -24674.29} C_VEL
LIN {X 0,Y 224.39,Z 497.525,A -85,B 0,C 180,E1 -24677.429,E2 -24677.429} C_VEL
LIN {X 0,Y 225.92,Z 500.7,A -85,B 0,C 180,E1 -24678.595,E2 -24678.595} C_VEL
LIN {X 0,Y 221.535,Z 545.515,A -85,B 0,C 180,E1 -24679.652,E2 -24679.652} C_VEL
LIN {X 0,Y 219.002,Z 561.177,A -85,B 0,C 180,E1 -24680.29,E2 -24680.29} C_VEL
LIN {X 0,Y 215.667,Z 574.625,A -85,B 0,C 180,E1 -24680.974,E2 -24680.974} C_VEL
LIN {X 0,Y 211.319,Z 588.686,A -85,B 0,C 180,E1 -24682.019,E2 -24682.019} C_VEL
LIN {X 0,Y 206.358,Z 601.243,A -85,B 0,C 180,E1 -24683.14,E2 -24683.14} C_VEL
LIN {X 0,Y 200.142,Z 614.785,A -85,B 0,C 180,E1 -24684.812,E2 -24684.812} C_VEL
LIN {X 0,Y 193.641,Z 626.659,A -85,B 0,C 180,E1 -24686.653,E2 -24686.653} C_VEL
LIN {X 0,Y 186.544,Z 637.839,A -85,B 0,C 180,E1 -24688.844,E2 -24688.844} C_VEL
LIN {X 0,Y 179.115,Z 648.102,A -85,B 0,C 180,E1 -24691.415,E2 -24691.415} C_VEL
LIN {X 0,Y 172.12,Z 656.769,A -85,B 0,C 180,E1 -24694.224,E2 -24694.224} C_VEL
LIN {X 0,Y 164.482,Z 665.219,A -85,B 0,C 180,E1 -24697.77,E2 -24697.77} C_VEL
LIN {X 0,Y 157.211,Z 672.531,A -85,B 0,C 180,E1 -24701.879,E2 -24701.879} C_VEL
LIN {X 0,Y 151.384,Z 677.866,A -85,B 0,C 180,E1 -24705.863,E2 -24705.863} C_VEL
LIN {X 0,Y 145.365,Z 682.955,A -85,B 0,C 180,E1 -24711.06,E2 -24711.06} C_VEL
LIN {X 0,Y 140.498,Z 686.671,A -85,B 0,C 180,E1 -24716.616,E2 -24716.616} C_VEL
LIN {X 0,Y 136.962,Z 689.119,A -85,B 0,C 180,E1 -24722.495,E2 -24722.495} C_VEL
LIN {X 0,Y 134.653,Z 690.345,A -85,B 0,C 180,E1 -24728.571,E2 -24728.571} C_VEL
LIN {X 0,Y 133.465,Z 690.358,A -85,B 0,C 180,E1 -24734.735,E2 -24734.735} C_VEL
LIN {X 0,Y 133.181,Z 689.225,A -85,B 0,C 180,E1 -24740.891,E2 -24740.891} C_VEL
LIN {X 0,Y 133.809,Z 686.94,A -85,B 0,C 180,E1 -24746.989,E2 -24746.989} C_VEL
LIN {X 0,Y 134.832,Z 683.491,A -85,B 0,C 180,E1 -24752.988,E2 -24752.988} C_VEL
LIN {X 0,Y 136.983,Z 678.777,A -85,B 0,C 180,E1 -24758.854,E2 -24758.854} C_VEL
LIN {X 0,Y 140.145,Z 672.688,A -85,B 0,C 180,E1 -24764.522,E2 -24764.522} C_VEL
LIN {X 0,Y 144.519,Z 665.023,A -85,B 0,C 180,E1 -24769.902,E2 -24769.902} C_VEL
LIN {X 0,Y 149.148,Z 656.861,A -85,B 0,C 180,E1 -24774.35,E2 -24774.35} C_VEL
LIN {X 0,Y 154.562,Z 647.047,A -85,B 0,C 180,E1 -24778.519,E2 -24778.519} C_VEL
LIN {X 0,Y 160.735,Z 635.157,A -85,B 0,C 180,E1 -24782.386,E2 -24782.386} C_VEL
LIN {X 0,Y 166.479,Z 622.821,A -85,B 0,C 180,E1 -24785.483,E2 -24785.483} C_VEL
LIN {X 0,Y 171.619,Z 610.47,A -85,B 0,C 180,E1 -24787.899,E2 -24787.899} C_VEL
LIN {X 0,Y 176.419,Z 596.972,A -85,B 0,C 180,E1 -24789.969,E2 -24789.969} C_VEL
LIN {X 0,Y 180.528,Z 582.995,A -85,B 0,C 180,E1 -24791.625,E2 -24791.625} C_VEL
LIN {X 0,Y 183.921,Z 568.616,A -85,B 0,C 180,E1 -24792.895,E2 -24792.895} C_VEL
LIN {X 0,Y 186.647,Z 552.727,A -85,B 0,C 180,E1 -24793.899,E2 -24793.899} C_VEL
LIN {X 0,Y 188.368,Z 536.645,A -85,B 0,C 180,E1 -24794.542,E2 -24794.542} C_VEL
LIN {X 0,Y 193.116,Z 475.509,A -85,B 0,C 180,E1 -24796.385,E2 -24796.385} C_VEL
LIN {X 0,Y 188.298,Z 465.472,A -85,B 0,C 180,E1 -24798.952,E2 -24798.952} C_VEL
LIN {X 0,Y 183.155,Z 456.167,A -85,B 0,C 180,E1 -24801.948,E2 -24801.948} C_VEL
LIN {X 0,Y 178.341,Z 448.045,A -85,B 0,C 180,E1 -24805.116,E2 -24805.116} C_VEL
LIN {X 0,Y 173.301,Z 440.345,A -85,B 0,C 180,E1 -24808.948,E2 -24808.948} C_VEL
LIN {X 0,Y 169.92,Z 435.635,A -85,B 0,C 180,E1 -24811.954,E2 -24811.954} C_VEL
LIN {X 0,Y 166.921,Z 431.454,A -85,B 0,C 180,E1 -24815.099,E2 -24815.099} C_VEL
LIN {X 0,Y 164.499,Z 428.402,A -85,B 0,C 180,E1 -24818.1,E2 -24818.1} C_VEL
LIN {X 0,Y 163.793,Z 426.954,A -85,B 0,C 180,E1 -24819.191,E2 -24819.191} C_VEL
LIN {X 0,Y 161.146,Z 424.425,A -85,B 0,C 180,E1 -24823.634,E2 -24823.634} C_VEL
LIN {X 0,Y 159.954,Z 421.547,A -85,B 0,C 180,E1 -24826.985,E2 -24826.985} C_VEL
LIN {X 0,Y 158.577,Z 420.83,A -85,B 0,C 180,E1 -24834.914,E2 -24834.914} C_VEL
LIN {X 0,Y 159.45,Z 421.076,A -85,B 0,C 180,E1 -24840.946,E2 -24840.946} C_VEL
LIN {X 0,Y 160.271,Z 421.694,A -85,B 0,C 180,E1 -24843.456,E2 -24843.456} C_VEL
LIN {X 0,Y 161.792,Z 424.863,A -85,B 0,C 180,E1 -24847.173,E2 -24847.173} C_VEL
LIN {X 0,Y 163.911,Z 427.041,A -85,B 0,C 180,E1 -24850.577,E2 -24850.577} C_VEL
LIN {X 0,Y 166.173,Z 430.642,A -85,B 0,C 180,E1 -24853.645,E2 -24853.645} C_VEL
LIN {X 0,Y 167.594,Z 432.237,A -85,B 0,C 180,E1 -24855.232,E2 -24855.232} C_VEL
LIN {X 0,Y 171.076,Z 437.19,A -85,B 0,C 180,E1 -24858.719,E2 -24858.719} C_VEL
LIN {X 0,Y 174.427,Z 442.086,A -85,B 0,C 180,E1 -24861.571,E2 -24861.571} C_VEL
LIN {X 0,Y 178.528,Z 448.306,A -85,B 0,C 180,E1 -24864.608,E2 -24864.608} C_VEL
LIN {X 0,Y 182.575,Z 455.047,A -85,B 0,C 180,E1 -24867.278,E2 -24867.278} C_VEL
LIN {X 0,Y 186.662,Z 464.239,A -85,B 0,C 180,E1 -24869.847,E2 -24869.847} C_VEL
LIN {X 0,Y 191.391,Z 476.594,A -85,B 0,C 180,E1 -24872.608,E2 -24872.608} C_VEL
LIN {X 0,Y 192.836,Z 480.665,A -85,B 0,C 180,E1 -24873.409,E2 -24873.409} C_VEL
LIN {X 0,Y 187.067,Z 553.411,A -85,B 0,C 180,E1 -24875.665,E2 -24875.665} C_VEL
LIN {X 0,Y 184.633,Z 569.397,A -85,B 0,C 180,E1 -24876.475,E2 -24876.475} C_VEL
LIN {X 0,Y 181.262,Z 584.607,A -85,B 0,C 180,E1 -24877.588,E2 -24877.588} C_VEL
LIN {X 0,Y 177.338,Z 598.348,A -85,B 0,C 180,E1 -24878.945,E2 -24878.945} C_VEL
LIN {X 0,Y 172.571,Z 612.585,A -85,B 0,C 180,E1 -24880.879,E2 -24880.879} C_VEL
LIN {X 0,Y 167.343,Z 625.588,A -85,B 0,C 180,E1 -24883.138,E2 -24883.138} C_VEL
LIN {X 0,Y 161.76,Z 638.038,A -85,B 0,C 180,E1 -24885.96,E2 -24885.96} C_VEL
LIN {X 0,Y 156.02,Z 649.361,A -85,B 0,C 180,E1 -24889.22,E2 -24889.22} C_VEL
LIN {X 0,Y 155.387,Z 650.567,A -85,B 0,C 180,E1 -24889.638,E2 -24889.638} C_VEL
LIN {X 0,Y 152.755,Z 654.615,A -85,B 0,C 180,E1 -24890.939,E2 -24890.939} C_VEL
LIN {X 0,Y 146.957,Z 660.77,A -85,B 0,C 180,E1 -24892.891,E2 -24892.891} C_VEL
LIN {X 0,Y 141.117,Z 666.566,A -85,B 0,C 180,E1 -24895.106,E2 -24895.106} C_VEL
LIN {X 0,Y 138.493,Z 669.863,A -85,B 0,C 180,E1 -24896.811,E2 -24896.811} C_VEL
LIN {X 0,Y 134.035,Z 677.483,A -85,B 0,C 180,E1 -24901.842,E2 -24901.842} C_VEL
LIN {X 0,Y 130.252,Z 684.369,A -85,B 0,C 180,E1 -24907.809,E2 -24907.809} C_VEL
LIN {X 0,Y 127.763,Z 689.759,A -85,B 0,C 180,E1 -24914.035,E2 -24914.035} C_VEL
LIN {X 0,Y 126.56,Z 693.767,A -85,B 0,C 180,E1 -24920.41,E2 -24920.41} C_VEL
LIN {X 0,Y 126.379,Z 696.485,A -85,B 0,C 180,E1 -24926.812,E2 -24926.812} C_VEL
LIN {X 0,Y 126.501,Z 697.383,A -85,B 0,C 180,E1 -24930,E2 -24930} C_VEL
LIN {X 0,Y 126.366,Z 697.973,A -85,B 0,C 180,E1 -24933.188,E2 -24933.188} C_VEL
LIN {X 0,Y 126.55,Z 698.297,A -85,B 0,C 180,E1 -24939.59,E2 -24939.59} C_VEL
LIN {X 0,Y 127.88,Z 697.51,A -85,B 0,C 180,E1 -24945.949,E2 -24945.949} C_VEL
LIN {X 0,Y 130.618,Z 695.549,A -85,B 0,C 180,E1 -24952.126,E2 -24952.126} C_VEL
LIN {X 0,Y 134.701,Z 692.439,A -85,B 0,C 180,E1 -24958.007,E2 -24958.007} C_VEL
LIN {X 0,Y 140.076,Z 688.123,A -85,B 0,C 180,E1 -24963.497,E2 -24963.497} C_VEL
LIN {X 0,Y 146.721,Z 682.49,A -85,B 0,C 180,E1 -24968.514,E2 -24968.514} C_VEL
LIN {X 0,Y 154.228,Z 675.396,A -85,B 0,C 180,E1 -24973.12,E2 -24973.12} C_VEL
LIN {X 0,Y 161.704,Z 667.85,A -85,B 0,C 180,E1 -24976.718,E2 -24976.718} C_VEL
LIN {X 0,Y 169.793,Z 658.803,A -85,B 0,C 180,E1 -24979.973,E2 -24979.973} C_VEL
LIN {X 0,Y 178.445,Z 647.909,A -85,B 0,C 180,E1 -24982.896,E2 -24982.896} C_VEL
LIN {X 0,Y 186.173,Z 636.757,A -85,B 0,C 180,E1 -24985.191,E2 -24985.191} C_VEL
LIN {X 0,Y 193.451,Z 624.553,A -85,B 0,C 180,E1 -24987.153,E2 -24987.153} C_VEL
LIN {X 0,Y 200.42,Z 611.119,A -85,B 0,C 180,E1 -24988.731,E2 -24988.731} C_VEL
LIN {X 0,Y 206.02,Z 597.964,A -85,B 0,C 180,E1 -24989.954,E2 -24989.954} C_VEL
LIN {X 0,Y 211.066,Z 583.57,A -85,B 0,C 180,E1 -24990.935,E2 -24990.935} C_VEL
LIN {X 0,Y 215.087,Z 568.684,A -85,B 0,C 180,E1 -24991.665,E2 -24991.665} C_VEL
LIN {X 0,Y 217.792,Z 554.301,A -85,B 0,C 180,E1 -24992.188,E2 -24992.188} C_VEL
LIN {X 0,Y 220.372,Z 530.941,A -85,B 0,C 180,E1 -24992.76,E2 -24992.76} C_VEL
LIN {X 0,Y 222.479,Z 508.394,A -85,B 0,C 180,E1 -24993.325,E2 -24993.325} C_VEL
LIN {X 0,Y 219.163,Z 499.3,A -85,B 0,C 180,E1 -24996.433,E2 -24996.433} C_VEL
LIN {X 0,Y 217.169,Z 494.458,A -85,B 0,C 180,E1 -24998.548,E2 -24998.548} C_VEL
LIN {X 0,Y 214.896,Z 489.212,A -85,B 0,C 180,E1 -25001.353,E2 -25001.353} C_VEL
LIN {X 0,Y 213.255,Z 486.171,A -85,B 0,C 180,E1 -25003.733,E2 -25003.733} C_VEL
LIN {X 0,Y 211.361,Z 482.556,A -85,B 0,C 180,E1 -25007.397,E2 -25007.397} C_VEL
LIN {X 0,Y 209.841,Z 479.586,A -85,B 0,C 180,E1 -25013.269,E2 -25013.269} C_VEL
LIN {X 0,Y 209.846,Z 478.451,A -85,B 0,C 180,E1 -25015.198,E2 -25015.198} C_VEL
LIN {X 0,Y 209.897,Z 478.438,A -85,B 0,C 180,E1 -25016.401,E2 -25016.401} C_VEL
LIN {X 0,Y 210.634,Z 481.596,A -85,B 0,C 180,E1 -25021.196,E2 -25021.196} C_VEL
LIN {X 0,Y 211.661,Z 482.895,A -85,B 0,C 180,E1 -25023.707,E2 -25023.707} C_VEL
LIN {X 0,Y 213.983,Z 487.311,A -85,B 0,C 180,E1 -25027.817,E2 -25027.817} C_VEL
LIN {X 0,Y 215.878,Z 490.818,A -85,B 0,C 180,E1 -25030.316,E2 -25030.316} C_VEL
LIN {X 0,Y 219.311,Z 497.493,A -85,B 0,C 180,E1 -25033.967,E2 -25033.967} C_VEL
LIN {X 0,Y 222.771,Z 504.452,A -85,B 0,C 180,E1 -25036.994,E2 -25036.994} C_VEL
LIN {X 0,Y 218.531,Z 546.689,A -85,B 0,C 180,E1 -25038.001,E2 -25038.001} C_VEL
LIN {X 0,Y 215.759,Z 562.604,A -85,B 0,C 180,E1 -25038.642,E2 -25038.642} C_VEL
LIN {X 0,Y 212.245,Z 576.215,A -85,B 0,C 180,E1 -25039.338,E2 -25039.338} C_VEL
LIN {X 0,Y 207.244,Z 591.427,A -85,B 0,C 180,E1 -25040.477,E2 -25040.477} C_VEL
LIN {X 0,Y 201.489,Z 605.105,A -85,B 0,C 180,E1 -25041.769,E2 -25041.769} C_VEL
LIN {X 0,Y 194.722,Z 618.704,A -85,B 0,C 180,E1 -25043.533,E2 -25043.533} C_VEL
LIN {X 0,Y 187.092,Z 631.447,A -85,B 0,C 180,E1 -25045.638,E2 -25045.638} C_VEL
LIN {X 0,Y 179.271,Z 642.715,A -85,B 0,C 180,E1 -25048.064,E2 -25048.064} C_VEL
LIN {X 0,Y 171.67,Z 652.285,A -85,B 0,C 180,E1 -25050.715,E2 -25050.715} C_VEL
LIN {X 0,Y 164.102,Z 660.832,A -85,B 0,C 180,E1 -25053.833,E2 -25053.833} C_VEL
LIN {X 0,Y 156.859,Z 668.188,A -85,B 0,C 180,E1 -25057.318,E2 -25057.318} C_VEL
LIN {X 0,Y 149.856,Z 674.672,A -85,B 0,C 180,E1 -25061.377,E2 -25061.377} C_VEL
LIN {X 0,Y 142.771,Z 680.571,A -85,B 0,C 180,E1 -25066.436,E2 -25066.436} C_VEL
LIN {X 0,Y 136.876,Z 685.026,A -85,B 0,C 180,E1 -25071.964,E2 -25071.964} C_VEL
LIN {X 0,Y 131.948,Z 688.36,A -85,B 0,C 180,E1 -25078.456,E2 -25078.456} C_VEL
LIN {X 0,Y 128.984,Z 690.047,A -85,B 0,C 180,E1 -25084.158,E2 -25084.158} C_VEL
LIN {X 0,Y 127.048,Z 690.704,A -85,B 0,C 180,E1 -25090.616,E2 -25090.616} C_VEL
LIN {X 0,Y 126.127,Z 690.205,A -85,B 0,C 180,E1 -25097.122,E2 -25097.122} C_VEL
LIN {X 0,Y 126.261,Z 688.559,A -85,B 0,C 180,E1 -25103.608,E2 -25103.608} C_VEL
LIN {X 0,Y 126.723,Z 687.299,A -85,B 0,C 180,E1 -25106.821,E2 -25106.821} C_VEL
LIN {X 0,Y 127.756,Z 683.916,A -85,B 0,C 180,E1 -25113.154,E2 -25113.154} C_VEL
LIN {X 0,Y 129.973,Z 679.269,A -85,B 0,C 180,E1 -25119.336,E2 -25119.336} C_VEL
LIN {X 0,Y 133.315,Z 673.24,A -85,B 0,C 180,E1 -25125.283,E2 -25125.283} C_VEL
LIN {X 0,Y 137.885,Z 665.663,A -85,B 0,C 180,E1 -25130.903,E2 -25130.903} C_VEL
LIN {X 0,Y 142.751,Z 657.554,A -85,B 0,C 180,E1 -25135.518,E2 -25135.518} C_VEL
LIN {X 0,Y 148.406,Z 647.838,A -85,B 0,C 180,E1 -25139.818,E2 -25139.818} C_VEL
LIN {X 0,Y 153.895,Z 637.886,A -85,B 0,C 180,E1 -25143.231,E2 -25143.231} C_VEL
LIN {X 0,Y 159.775,Z 626.077,A -85,B 0,C 180,E1 -25146.429,E2 -25146.429} C_VEL
LIN {X 0,Y 165.049,Z 614.293,A -85,B 0,C 180,E1 -25148.909,E2 -25148.909} C_VEL
LIN {X 0,Y 169.976,Z 601.583,A -85,B 0,C 180,E1 -25151.025,E2 -25151.025} C_VEL
LIN {X 0,Y 174.5,Z 587.701,A -85,B 0,C 180,E1 -25152.816,E2 -25152.816} C_VEL
LIN {X 0,Y 178.219,Z 573.4,A -85,B 0,C 180,E1 -25154.227,E2 -25154.227} C_VEL
LIN {X 0,Y 181.175,Z 558.765,A -85,B 0,C 180,E1 -25155.264,E2 -25155.264} C_VEL
LIN {X 0,Y 183.21,Z 543.979,A -85,B 0,C 180,E1 -25155.99,E2 -25155.99} C_VEL
LIN {X 0,Y 188.606,Z 478.351,A -85,B 0,C 180,E1 -25157.998,E2 -25157.998} C_VEL
LIN {X 0,Y 183.716,Z 468.036,A -85,B 0,C 180,E1 -25160.836,E2 -25160.836} C_VEL
LIN {X 0,Y 177.636,Z 456.977,A -85,B 0,C 180,E1 -25164.796,E2 -25164.796} C_VEL
LIN {X 0,Y 172.764,Z 449.134,A -85,B 0,C 180,E1 -25168.489,E2 -25168.489} C_VEL
LIN {X 0,Y 170.039,Z 445.054,A -85,B 0,C 180,E1 -25170.859,E2 -25170.859} C_VEL
LIN {X 0,Y 168.071,Z 442.043,A -85,B 0,C 180,E1 -25172.782,E2 -25172.782} C_VEL
LIN {X 0,Y 165.305,Z 438.089,A -85,B 0,C 180,E1 -25175.844,E2 -25175.844} C_VEL
LIN {X 0,Y 162.839,Z 434.621,A -85,B 0,C 180,E1 -25179.155,E2 -25179.155} C_VEL
LIN {X 0,Y 162.176,Z 433.582,A -85,B 0,C 180,E1 -25180.206,E2 -25180.206} C_VEL
LIN {X 0,Y 159.689,Z 430.703,A -85,B 0,C 180,E1 -25184.933,E2 -25184.933} C_VEL
LIN {X 0,Y 158.982,Z 428.62,A -85,B 0,C 180,E1 -25187.229,E2 -25187.229} C_VEL
LIN {X 0,Y 157.709,Z 427.858,A -85,B 0,C 180,E1 -25194.886,E2 -25194.886} C_VEL
LIN {X 0,Y 158.575,Z 428.128,A -85,B 0,C 180,E1 -25200.951,E2 -25200.951} C_VEL
LIN {X 0,Y 159.217,Z 428.657,A -85,B 0,C 180,E1 -25203.004,E2 -25203.004} C_VEL
LIN {X 0,Y 160.627,Z 431.732,A -85,B 0,C 180,E1 -25206.673,E2 -25206.673} C_VEL
LIN {X 0,Y 162.557,Z 433.853,A -85,B 0,C 180,E1 -25209.958,E2 -25209.958} C_VEL
LIN {X 0,Y 164.887,Z 437.547,A -85,B 0,C 180,E1 -25213.243,E2 -25213.243} C_VEL
LIN {X 0,Y 166.004,Z 438.954,A -85,B 0,C 180,E1 -25214.558,E2 -25214.558} C_VEL
LIN {X 0,Y 169.285,Z 443.793,A -85,B 0,C 180,E1 -25218.013,E2 -25218.013} C_VEL
LIN {X 0,Y 172.479,Z 448.63,A -85,B 0,C 180,E1 -25220.864,E2 -25220.864} C_VEL
LIN {X 0,Y 176.343,Z 454.823,A -85,B 0,C 180,E1 -25223.876,E2 -25223.876} C_VEL
LIN {X 0,Y 179.749,Z 460.771,A -85,B 0,C 180,E1 -25226.25,E2 -25226.25} C_VEL
LIN {X 0,Y 183.409,Z 469.502,A -85,B 0,C 180,E1 -25228.716,E2 -25228.716} C_VEL
LIN {X 0,Y 187.619,Z 480.939,A -85,B 0,C 180,E1 -25231.351,E2 -25231.351} C_VEL
LIN {X 0,Y 188.304,Z 482.897,A -85,B 0,C 180,E1 -25231.76,E2 -25231.76} C_VEL
LIN {X 0,Y 183.38,Z 544.877,A -85,B 0,C 180,E1 -25233.657,E2 -25233.657} C_VEL
LIN {X 0,Y 181.573,Z 560.583,A -85,B 0,C 180,E1 -25234.296,E2 -25234.296} C_VEL
LIN {X 0,Y 178.6,Z 576.363,A -85,B 0,C 180,E1 -25235.261,E2 -25235.261} C_VEL
LIN {X 0,Y 174.781,Z 590.88,A -85,B 0,C 180,E1 -25236.466,E2 -25236.466} C_VEL
LIN {X 0,Y 170.547,Z 604.171,A -85,B 0,C 180,E1 -25237.99,E2 -25237.99} C_VEL
LIN {X 0,Y 165.341,Z 617.994,A -85,B 0,C 180,E1 -25240.083,E2 -25240.083} C_VEL
LIN {X 0,Y 159.814,Z 630.586,A -85,B 0,C 180,E1 -25242.557,E2 -25242.557} C_VEL
LIN {X 0,Y 153.583,Z 643.14,A -85,B 0,C 180,E1 -25245.745,E2 -25245.745} C_VEL
LIN {X 0,Y 147.972,Z 653.432,A -85,B 0,C 180,E1 -25249.139,E2 -25249.139} C_VEL
LIN {X 0,Y 142.123,Z 663.838,A -85,B 0,C 180,E1 -25253.601,E2 -25253.601} C_VEL
LIN {X 0,Y 138.493,Z 669.863,A -85,B 0,C 180,E1 -25256.811,E2 -25256.811} C_VEL
LIN {X 0,Y 135.957,Z 673.05,A -85,B 0,C 180,E1 -25258.621,E2 -25258.621} C_VEL
LIN {X 0,Y 130.487,Z 677.787,A -85,B 0,C 180,E1 -25261.525,E2 -25261.525} C_VEL
LIN {X 0,Y 125.314,Z 682.084,A -85,B 0,C 180,E1 -25264.789,E2 -25264.789} C_VEL
LIN {X 0,Y 123.328,Z 684.431,A -85,B 0,C 180,E1 -25267.115,E2 -25267.115} C_VEL
LIN {X 0,Y 120.884,Z 689.354,A -85,B 0,C 180,E1 -25273.1,E2 -25273.1} C_VEL
LIN {X 0,Y 119.51,Z 693.406,A -85,B 0,C 180,E1 -25279.838,E2 -25279.838} C_VEL
LIN {X 0,Y 119.279,Z 696.178,A -85,B 0,C 180,E1 -25286.622,E2 -25286.622} C_VEL
LIN {X 0,Y 119.414,Z 697.103,A -85,B 0,C 180,E1 -25290,E2 -25290} C_VEL
LIN {X 0,Y 119.269,Z 697.716,A -85,B 0,C 180,E1 -25293.378,E2 -25293.378} C_VEL
LIN {X 0,Y 119.534,Z 698.09,A -85,B 0,C 180,E1 -25300.159,E2 -25300.159} C_VEL
LIN {X 0,Y 121.009,Z 697.339,A -85,B 0,C 180,E1 -25306.881,E2 -25306.881} C_VEL
LIN {X 0,Y 124.006,Z 695.418,A -85,B 0,C 180,E1 -25313.373,E2 -25313.373} C_VEL
LIN {X 0,Y 128.438,Z 692.361,A -85,B 0,C 180,E1 -25319.503,E2 -25319.503} C_VEL
LIN {X 0,Y 134.165,Z 688.101,A -85,B 0,C 180,E1 -25325.185,E2 -25325.185} C_VEL
LIN {X 0,Y 141.204,Z 682.528,A -85,B 0,C 180,E1 -25330.318,E2 -25330.318} C_VEL
LIN {X 0,Y 149.084,Z 675.499,A -85,B 0,C 180,E1 -25335.001,E2 -25335.001} C_VEL
LIN {X 0,Y 156.903,Z 668.02,A -85,B 0,C 180,E1 -25338.614,E2 -25338.614} C_VEL
LIN {X 0,Y 165.31,Z 659.029,A -85,B 0,C 180,E1 -25341.86,E2 -25341.86} C_VEL
LIN {X 0,Y 174.258,Z 648.251,A -85,B 0,C 180,E1 -25344.756,E2 -25344.756} C_VEL
LIN {X 0,Y 182.907,Z 636.182,A -85,B 0,C 180,E1 -25347.195,E2 -25347.195} C_VEL
LIN {X 0,Y 189.708,Z 625.107,A -85,B 0,C 180,E1 -25348.948,E2 -25348.948} C_VEL
LIN {X 0,Y 196.849,Z 611.843,A -85,B 0,C 180,E1 -25350.488,E2 -25350.488} C_VEL
LIN {X 0,Y 201.839,Z 600.658,A -85,B 0,C 180,E1 -25351.546,E2 -25351.546} C_VEL
LIN {X 0,Y 207.383,Z 585.94,A -85,B 0,C 180,E1 -25352.557,E2 -25352.557} C_VEL
LIN {X 0,Y 211.643,Z 571.219,A -85,B 0,C 180,E1 -25353.313,E2 -25353.313} C_VEL
LIN {X 0,Y 214.877,Z 555.656,A -85,B 0,C 180,E1 -25353.861,E2 -25353.861} C_VEL
LIN {X 0,Y 217.29,Z 535.319,A -85,B 0,C 180,E1 -25354.383,E2 -25354.383} C_VEL
LIN {X 0,Y 219.548,Z 511.886,A -85,B 0,C 180,E1 -25354.959,E2 -25354.959} C_VEL
LIN {X 0,Y 216.648,Z 503.616,A -85,B 0,C 180,E1 -25357.985,E2 -25357.985} C_VEL
LIN {X 0,Y 214.286,Z 497.739,A -85,B 0,C 180,E1 -25360.855,E2 -25360.855} C_VEL
LIN {X 0,Y 213.294,Z 495.408,A -85,B 0,C 180,E1 -25362.255,E2 -25362.255} C_VEL
LIN {X 0,Y 212.09,Z 493.01,A -85,B 0,C 180,E1 -25364.135,E2 -25364.135} C_VEL
LIN {X 0,Y 210.343,Z 489.49,A -85,B 0,C 180,E1 -25367.702,E2 -25367.702} C_VEL
LIN {X 0,Y 208.949,Z 486.594,A -85,B 0,C 180,E1 -25373.483,E2 -25373.483} C_VEL
LIN {X 0,Y 208.973,Z 485.528,A -85,B 0,C 180,E1 -25375.178,E2 -25375.178} C_VEL
LIN {X 0,Y 209.012,Z 485.594,A -85,B 0,C 180,E1 -25376.386,E2 -25376.386} C_VEL
LIN {X 0,Y 209.677,Z 488.578,A -85,B 0,C 180,E1 -25380.961,E2 -25380.961} C_VEL
LIN {X 0,Y 210.618,Z 489.876,A -85,B 0,C 180,E1 -25383.393,E2 -25383.393} C_VEL
LIN {X 0,Y 212.846,Z 494.282,A -85,B 0,C 180,E1 -25387.511,E2 -25387.511} C_VEL
LIN {X 0,Y 214.725,Z 498.018,A -85,B 0,C 180,E1 -25390.089,E2 -25390.089} C_VEL
LIN {X 0,Y 218.231,Z 505.137,A -85,B 0,C 180,E1 -25393.904,E2 -25393.904} C_VEL
LIN {X 0,Y 219.818,Z 508.527,A -85,B 0,C 180,E1 -25395.387,E2 -25395.387} C_VEL
LIN {X 0,Y 215.832,Z 546.89,A -85,B 0,C 180,E1 -25396.273,E2 -25396.273} C_VEL
LIN {X 0,Y 213.002,Z 562.731,A -85,B 0,C 180,E1 -25396.892,E2 -25396.892} C_VEL
LIN {X 0,Y 209.282,Z 576.806,A -85,B 0,C 180,E1 -25397.593,E2 -25397.593} C_VEL
LIN {X 0,Y 204.07,Z 592.126,A -85,B 0,C 180,E1 -25398.724,E2 -25398.724} C_VEL
LIN {X 0,Y 198.171,Z 605.72,A -85,B 0,C 180,E1 -25399.981,E2 -25399.981} C_VEL
LIN {X 0,Y 191.255,Z 619.152,A -85,B 0,C 180,E1 -25401.694,E2 -25401.694} C_VEL
LIN {X 0,Y 184.056,Z 630.906,A -85,B 0,C 180,E1 -25403.592,E2 -25403.592} C_VEL
LIN {X 0,Y 176.454,Z 641.581,A -85,B 0,C 180,E1 -25405.791,E2 -25405.791} C_VEL
LIN {X 0,Y 168.049,Z 651.93,A -85,B 0,C 180,E1 -25408.568,E2 -25408.568} C_VEL
LIN {X 0,Y 159.413,Z 661.313,A -85,B 0,C 180,E1 -25411.942,E2 -25411.942} C_VEL
LIN {X 0,Y 151.391,Z 669.039,A -85,B 0,C 180,E1 -25415.669,E2 -25415.669} C_VEL
LIN {X 0,Y 145.081,Z 674.58,A -85,B 0,C 180,E1 -25419.189,E2 -25419.189} C_VEL
LIN {X 0,Y 137.518,Z 680.552,A -85,B 0,C 180,E1 -25424.317,E2 -25424.317} C_VEL
LIN {X 0,Y 131.141,Z 685.076,A -85,B 0,C 180,E1 -25429.977,E2 -25429.977} C_VEL
LIN {X 0,Y 126.101,Z 688.274,A -85,B 0,C 180,E1 -25436.129,E2 -25436.129} C_VEL
LIN {X 0,Y 122.4,Z 690.195,A -85,B 0,C 180,E1 -25442.655,E2 -25442.655} C_VEL
LIN {X 0,Y 120.181,Z 690.913,A -85,B 0,C 180,E1 -25449.459,E2 -25449.459} C_VEL
LIN {X 0,Y 119.075,Z 690.475,A -85,B 0,C 180,E1 -25456.344,E2 -25456.344} C_VEL
LIN {X 0,Y 119.139,Z 688.889,A -85,B 0,C 180,E1 -25463.225,E2 -25463.225} C_VEL
LIN {X 0,Y 119.641,Z 687.489,A -85,B 0,C 180,E1 -25467.025,E2 -25467.025} C_VEL
LIN {X 0,Y 120.683,Z 684.34,A -85,B 0,C 180,E1 -25473.339,E2 -25473.339} C_VEL
LIN {X 0,Y 122.973,Z 679.741,A -85,B 0,C 180,E1 -25479.872,E2 -25479.872} C_VEL
LIN {X 0,Y 126.512,Z 673.769,A -85,B 0,C 180,E1 -25486.127,E2 -25486.127} C_VEL
LIN {X 0,Y 131.3,Z 666.272,A -85,B 0,C 180,E1 -25492.005,E2 -25492.005} C_VEL
LIN {X 0,Y 136.421,Z 658.24,A -85,B 0,C 180,E1 -25496.794,E2 -25496.794} C_VEL
LIN {X 0,Y 142.334,Z 648.617,A -85,B 0,C 180,E1 -25501.229,E2 -25501.229} C_VEL
LIN {X 0,Y 148.041,Z 638.779,A -85,B 0,C 180,E1 -25504.728,E2 -25504.728} C_VEL
LIN {X 0,Y 154.169,Z 627.102,A -85,B 0,C 180,E1 -25507.982,E2 -25507.982} C_VEL
LIN {X 0,Y 160.195,Z 614.205,A -85,B 0,C 180,E1 -25510.737,E2 -25510.737} C_VEL
LIN {X 0,Y 165.314,Z 601.427,A -85,B 0,C 180,E1 -25512.86,E2 -25512.86} C_VEL
LIN {X 0,Y 170,Z 587.451,A -85,B 0,C 180,E1 -25514.652,E2 -25514.652} C_VEL
LIN {X 0,Y 173.875,Z 572.999,A -85,B 0,C 180,E1 -25516.053,E2 -25516.053} C_VEL
LIN {X 0,Y 177.076,Z 557.205,A -85,B 0,C 180,E1 -25517.14,E2 -25517.14} C_VEL
LIN {X 0,Y 179.15,Z 541.297,A -85,B 0,C 180,E1 -25517.876,E2 -25517.876} C_VEL
LIN {X 0,Y 184.231,Z 481.087,A -85,B 0,C 180,E1 -25519.704,E2 -25519.704} C_VEL
LIN {X 0,Y 179.558,Z 471.288,A -85,B 0,C 180,E1 -25522.649,E2 -25522.649} C_VEL
LIN {X 0,Y 174.424,Z 461.733,A -85,B 0,C 180,E1 -25526.292,E2 -25526.292} C_VEL
LIN {X 0,Y 170.275,Z 454.821,A -85,B 0,C 180,E1 -25529.692,E2 -25529.692} C_VEL
LIN {X 0,Y 166.658,Z 448.969,A -85,B 0,C 180,E1 -25533.21,E2 -25533.21} C_VEL
LIN {X 0,Y 163.707,Z 444.684,A -85,B 0,C 180,E1 -25536.621,E2 -25536.621} C_VEL
LIN {X 0,Y 161.306,Z 441.036,A -85,B 0,C 180,E1 -25540.094,E2 -25540.094} C_VEL
LIN {X 0,Y 160.608,Z 440.209,A -85,B 0,C 180,E1 -25541.24,E2 -25541.24} C_VEL
LIN {X 0,Y 158.253,Z 436.767,A -85,B 0,C 180,E1 -25546.473,E2 -25546.473} C_VEL
LIN {X 0,Y 157.872,Z 435.526,A -85,B 0,C 180,E1 -25547.952,E2 -25547.952} C_VEL
LIN {X 0,Y 156.839,Z 434.905,A -85,B 0,C 180,E1 -25554.857,E2 -25554.857} C_VEL
LIN {X 0,Y 157.7,Z 435.18,A -85,B 0,C 180,E1 -25560.956,E2 -25560.956} C_VEL
LIN {X 0,Y 158.169,Z 435.645,A -85,B 0,C 180,E1 -25562.546,E2 -25562.546} C_VEL
LIN {X 0,Y 159.641,Z 438.829,A -85,B 0,C 180,E1 -25566.516,E2 -25566.516} C_VEL
LIN {X 0,Y 161.199,Z 440.632,A -85,B 0,C 180,E1 -25569.29,E2 -25569.29} C_VEL
LIN {X 0,Y 163.758,Z 444.62,A -85,B 0,C 180,E1 -25573.02,E2 -25573.02} C_VEL
LIN {X 0,Y 167.443,Z 450.249,A -85,B 0,C 180,E1 -25577.21,E2 -25577.21} C_VEL
LIN {X 0,Y 171.409,Z 456.445,A -85,B 0,C 180,E1 -25580.866,E2 -25580.866} C_VEL
LIN {X 0,Y 176.455,Z 465.274,A -85,B 0,C 180,E1 -25584.799,E2 -25584.799} C_VEL
LIN {X 0,Y 180.016,Z 474.043,A -85,B 0,C 180,E1 -25587.383,E2 -25587.383} C_VEL
LIN {X 0,Y 184.01,Z 485.43,A -85,B 0,C 180,E1 -25590.084,E2 -25590.084} C_VEL
LIN {X 0,Y 178.275,Z 552.755,A -85,B 0,C 180,E1 -25592.171,E2 -25592.171} C_VEL
LIN {X 0,Y 175.835,Z 568.116,A -85,B 0,C 180,E1 -25592.927,E2 -25592.927} C_VEL
LIN {X 0,Y 172.248,Z 583.55,A -85,B 0,C 180,E1 -25594.026,E2 -25594.026} C_VEL
LIN {X 0,Y 168.065,Z 597.409,A -85,B 0,C 180,E1 -25595.369,E2 -25595.369} C_VEL
LIN {X 0,Y 163.068,Z 611.366,A -85,B 0,C 180,E1 -25597.237,E2 -25597.237} C_VEL
LIN {X 0,Y 157.288,Z 624.824,A -85,B 0,C 180,E1 -25599.576,E2 -25599.576} C_VEL
LIN {X 0,Y 151.189,Z 637.329,A -85,B 0,C 180,E1 -25602.443,E2 -25602.443} C_VEL
LIN {X 0,Y 144.443,Z 649.538,A -85,B 0,C 180,E1 -25606.104,E2 -25606.104} C_VEL
LIN {X 0,Y 138.919,Z 659.018,A -85,B 0,C 180,E1 -25609.832,E2 -25609.832} C_VEL
LIN {X 0,Y 133.194,Z 668.283,A -85,B 0,C 180,E1 -25614.52,E2 -25614.52} C_VEL
LIN {X 0,Y 128.34,Z 675.956,A -85,B 0,C 180,E1 -25619.566,E2 -25619.566} C_VEL
LIN {X 0,Y 124.655,Z 682.001,A -85,B 0,C 180,E1 -25624.674,E2 -25624.674} C_VEL
LIN {X 0,Y 123.328,Z 684.431,A -85,B 0,C 180,E1 -25627.115,E2 -25627.115} C_VEL
LIN {X 0,Y 121.497,Z 686.661,A -85,B 0,C 180,E1 -25629.547,E2 -25629.547} C_VEL
LIN {X 0,Y 117.168,Z 689.792,A -85,B 0,C 180,E1 -25633.562,E2 -25633.562} C_VEL
LIN {X 0,Y 113.927,Z 691.932,A -85,B 0,C 180,E1 -25637.016,E2 -25637.016} C_VEL
LIN {X 0,Y 112.476,Z 693.369,A -85,B 0,C 180,E1 -25639.843,E2 -25639.843} C_VEL
LIN {X 0,Y 112.299,Z 693.751,A -85,B 0,C 180,E1 -25640.822,E2 -25640.822} C_VEL
LIN {X 0,Y 112.167,Z 695.869,A -85,B 0,C 180,E1 -25646.407,E2 -25646.407} C_VEL
LIN {X 0,Y 112.329,Z 696.821,A -85,B 0,C 180,E1 -25650,E2 -25650} C_VEL
LIN {X 0,Y 112.175,Z 697.809,A -85,B 0,C 180,E1 -25657.198,E2 -25657.198} C_VEL
LIN {X 0,Y 113.17,Z 697.673,A -85,B 0,C 180,E1 -25664.383,E2 -25664.383} C_VEL
LIN {X 0,Y 115.659,Z 696.362,A -85,B 0,C 180,E1 -25671.382,E2 -25671.382} C_VEL
LIN {X 0,Y 119.932,Z 693.725,A -85,B 0,C 180,E1 -25678.481,E2 -25678.481} C_VEL
LIN {X 0,Y 125.179,Z 690.338,A -85,B 0,C 180,E1 -25684.155,E2 -25684.155} C_VEL
LIN {X 0,Y 131.916,Z 685.495,A -85,B 0,C 180,E1 -25689.741,E2 -25689.741} C_VEL
LIN {X 0,Y 139.876,Z 679.277,A -85,B 0,C 180,E1 -25694.702,E2 -25694.702} C_VEL
LIN {X 0,Y 147.562,Z 672.585,A -85,B 0,C 180,E1 -25698.602,E2 -25698.602} C_VEL
LIN {X 0,Y 155.993,Z 664.526,A -85,B 0,C 180,E1 -25702.039,E2 -25702.039} C_VEL
LIN {X 0,Y 164.924,Z 654.898,A -85,B 0,C 180,E1 -25705.116,E2 -25705.116} C_VEL
LIN {X 0,Y 172.982,Z 645.091,A -85,B 0,C 180,E1 -25707.463,E2 -25707.463} C_VEL
LIN {X 0,Y 181.202,Z 633.616,A -85,B 0,C 180,E1 -25709.582,E2 -25709.582} C_VEL
LIN {X 0,Y 186.157,Z 625.66,A -85,B 0,C 180,E1 -25710.814,E2 -25710.814} C_VEL
LIN {X 0,Y 193.47,Z 612.561,A -85,B 0,C 180,E1 -25712.307,E2 -25712.307} C_VEL
LIN {X 0,Y 199.33,Z 599.844,A -85,B 0,C 180,E1 -25713.467,E2 -25713.467} C_VEL
LIN {X 0,Y 204.982,Z 584.966,A -85,B 0,C 180,E1 -25714.442,E2 -25714.442} C_VEL
LIN {X 0,Y 209.331,Z 570.06,A -85,B 0,C 180,E1 -25715.15,E2 -25715.15} C_VEL
LIN {X 0,Y 212.402,Z 555.175,A -85,B 0,C 180,E1 -25715.67,E2 -25715.67} C_VEL
LIN {X 0,Y 214.912,Z 534.544,A -85,B 0,C 180,E1 -25716.165,E2 -25716.165} C_VEL
